Universal Robots URScript: draw_logo.script

def draw_image():
    # Get current TCP pose as starting reference (center of A4 paper)
    pose0 = get_actual_tcp_pose()
    x_c = pose0[0]
    y_c = pose0[1]
    z_c = pose0[2]
    rx  = pose0[3]
    ry  = pose0[4]
    rz  = pose0[5]

    # Movement parameters
    a = 0.3      # acceleration
    v = 0.05     # velocity
    z_lift = 0.01  # lift height between paths

    # A4 paper dimensions: 0.21m x 0.297m
    # SVG dimensions: 268.65231 x 393.11508

    # --- Path segment 1 ---
    # Move to start of segment (pen up)
    movel(p[x_c + -0.029184, y_c + -0.124246, z_c + z_lift, rx, ry, rz], a, v)
    # Lower pen
    movel(p[x_c + -0.029184, y_c + -0.124246, z_c, rx, ry, rz], a, v)

    # Draw path
    movel(p[x_c + -0.029184, y_c + -0.124246, z_c, rx, ry, rz], a, v)
    movel(p[x_c + -0.029184, y_c + -0.124246, z_c, rx, ry, rz], a, v)
    movel(p[x_c + -0.029184, y_c + -0.124246, z_c, rx, ry, rz], a, v)
    movel(p[x_c + -0.029184, y_c + -0.124246, z_c, rx, ry, rz], a, v)
    movel(p[x_c + -0.029184, y_c + -0.124246, z_c, rx, ry, rz], a, v)
    movel(p[x_c + -0.029184, y_c + -0.124246, z_c, rx, ry, rz], a, v)
    movel(p[x_c + -0.029184, y_c + -0.124246, z_c, rx, ry, rz], a, v)
    movel(p[x_c + -0.029184, y_c + -0.124246, z_c, rx, ry, rz], a, v)
    movel(p[x_c + -0.029184, y_c + -0.124246, z_c, rx, ry, rz], a, v)
    movel(p[x_c + -0.029184, y_c + -0.124246, z_c, rx, ry, rz], a, v)
    movel(p[x_c + -0.029182, y_c + -0.124228, z_c, rx, ry, rz], a, v)
    movel(p[x_c + -0.029174, y_c + -0.124205, z_c, rx, ry, rz], a, v)
    movel(p[x_c + -0.029161, y_c + -0.124179, z_c, rx, ry, rz], a, v)
    movel(p[x_c + -0.029143, y_c + -0.124148, z_c, rx, ry, rz], a, v)
    movel(p[x_c + -0.029120, y_c + -0.124114, z_c, rx, ry, rz], a, v)
    movel(p[x_c + -0.029093, y_c + -0.124076, z_c, rx, ry, rz], a, v)
    movel(p[x_c + -0.029062, y_c + -0.124034, z_c, rx, ry, rz], a, v)
    movel(p[x_c + -0.029026, y_c + -0.123989, z_c, rx, ry, rz], a, v)
    movel(p[x_c + -0.028986, y_c + -0.123941, z_c, rx, ry, rz], a, v)
    movel(p[x_c + -0.028943, y_c + -0.123889, z_c, rx, ry, rz], a, v)
    movel(p[x_c + -0.028896, y_c + -0.123835, z_c, rx, ry, rz], a, v)
    movel(p[x_c + -0.028845, y_c + -0.123778, z_c, rx, ry, rz], a, v)
    movel(p[x_c + -0.028791, y_c + -0.123719, z_c, rx, ry, rz], a, v)
    movel(p[x_c + -0.028734, y_c + -0.123657, z_c, rx, ry, rz], a, v)
    movel(p[x_c + -0.028674, y_c + -0.123593, z_c, rx, ry, rz], a, v)
    movel(p[x_c + -0.028610, y_c + -0.123527, z_c, rx, ry, rz], a, v)
    movel(p[x_c + -0.028545, y_c + -0.123459, z_c, rx, ry, rz], a, v)
    movel(p[x_c + -0.028477, y_c + -0.123389, z_c, rx, ry, rz], a, v)
    movel(p[x_c + -0.028406, y_c + -0.123318, z_c, rx, ry, rz], a, v)
    movel(p[x_c + -0.028334, y_c + -0.123245, z_c, rx, ry, rz], a, v)
    movel(p[x_c + -0.028259, y_c + -0.123171, z_c, rx, ry, rz], a, v)
    movel(p[x_c + -0.028183, y_c + -0.123096, z_c, rx, ry, rz], a, v)
    movel(p[x_c + -0.028105, y_c + -0.123021, z_c, rx, ry, rz], a, v)
    movel(p[x_c + -0.028025, y_c + -0.122944, z_c, rx, ry, rz], a, v)
    movel(p[x_c + -0.027945, y_c + -0.122867, z_c, rx, ry, rz], a, v)
    movel(p[x_c + -0.027863, y_c + -0.122789, z_c, rx, ry, rz], a, v)
    movel(p[x_c + -0.027780, y_c + -0.122711, z_c, rx, ry, rz], a, v)
    movel(p[x_c + -0.027697, y_c + -0.122634, z_c, rx, ry, rz], a, v)
    movel(p[x_c + -0.027613, y_c + -0.122556, z_c, rx, ry, rz], a, v)
    movel(p[x_c + -0.027528, y_c + -0.122478, z_c, rx, ry, rz], a, v)
    movel(p[x_c + -0.027444, y_c + -0.122401, z_c, rx, ry, rz], a, v)
    movel(p[x_c + -0.027359, y_c + -0.122324, z_c, rx, ry, rz], a, v)
    movel(p[x_c + -0.027274, y_c + -0.122249, z_c, rx, ry, rz], a, v)
    movel(p[x_c + -0.027190, y_c + -0.122174, z_c, rx, ry, rz], a, v)
    movel(p[x_c + -0.027106, y_c + -0.122100, z_c, rx, ry, rz], a, v)
    movel(p[x_c + -0.027023, y_c + -0.122027, z_c, rx, ry, rz], a, v)
    movel(p[x_c + -0.026940, y_c + -0.121956, z_c, rx, ry, rz], a, v)
    movel(p[x_c + -0.026858, y_c + -0.121886, z_c, rx, ry, rz], a, v)
    movel(p[x_c + -0.026778, y_c + -0.121819, z_c, rx, ry, rz], a, v)
    movel(p[x_c + -0.026699, y_c + -0.121753, z_c, rx, ry, rz], a, v)
    movel(p[x_c + -0.026621, y_c + -0.121689, z_c, rx, ry, rz], a, v)
    movel(p[x_c + -0.026545, y_c + -0.121627, z_c, rx, ry, rz], a, v)
    movel(p[x_c + -0.026471, y_c + -0.121568, z_c, rx, ry, rz], a, v)
    movel(p[x_c + -0.026399, y_c + -0.121511, z_c, rx, ry, rz], a, v)
    movel(p[x_c + -0.026329, y_c + -0.121457, z_c, rx, ry, rz], a, v)
    movel(p[x_c + -0.026261, y_c + -0.121406, z_c, rx, ry, rz], a, v)
    movel(p[x_c + -0.026196, y_c + -0.121357, z_c, rx, ry, rz], a, v)
    movel(p[x_c + -0.026134, y_c + -0.121313, z_c, rx, ry, rz], a, v)
    movel(p[x_c + -0.026074, y_c + -0.121271, z_c, rx, ry, rz], a, v)
    movel(p[x_c + -0.026074, y_c + -0.121271, z_c, rx, ry, rz], a, v)
    movel(p[x_c + -0.025308, y_c + -0.120746, z_c, rx, ry, rz], a, v)
    movel(p[x_c + -0.025308, y_c + -0.120746, z_c, rx, ry, rz], a, v)
    movel(p[x_c + -0.025963, y_c + -0.120548, z_c, rx, ry, rz], a, v)
    movel(p[x_c + -0.025963, y_c + -0.120548, z_c, rx, ry, rz], a, v)
    movel(p[x_c + -0.026039, y_c + -0.120528, z_c, rx, ry, rz], a, v)
    movel(p[x_c + -0.026135, y_c + -0.120508, z_c, rx, ry, rz], a, v)
    movel(p[x_c + -0.026248, y_c + -0.120489, z_c, rx, ry, rz], a, v)
    movel(p[x_c + -0.026379, y_c + -0.120471, z_c, rx, ry, rz], a, v)
    movel(p[x_c + -0.026527, y_c + -0.120453, z_c, rx, ry, rz], a, v)
    movel(p[x_c + -0.026690, y_c + -0.120435, z_c, rx, ry, rz], a, v)
    movel(p[x_c + -0.026869, y_c + -0.120418, z_c, rx, ry, rz], a, v)
    movel(p[x_c + -0.027061, y_c + -0.120402, z_c, rx, ry, rz], a, v)
    movel(p[x_c + -0.027268, y_c + -0.120386, z_c, rx, ry, rz], a, v)
    movel(p[x_c + -0.027487, y_c + -0.120371, z_c, rx, ry, rz], a, v)
    movel(p[x_c + -0.027718, y_c + -0.120357, z_c, rx, ry, rz], a, v)
    movel(p[x_c + -0.027961, y_c + -0.120343, z_c, rx, ry, rz], a, v)
    movel(p[x_c + -0.028214, y_c + -0.120330, z_c, rx, ry, rz], a, v)
    movel(p[x_c + -0.028477, y_c + -0.120317, z_c, rx, ry, rz], a, v)
    movel(p[x_c + -0.028748, y_c + -0.120305, z_c, rx, ry, rz], a, v)
    movel(p[x_c + -0.029028, y_c + -0.120294, z_c, rx, ry, rz], a, v)
    movel(p[x_c + -0.029316, y_c + -0.120283, z_c, rx, ry, rz], a, v)
    movel(p[x_c + -0.029610, y_c + -0.120273, z_c, rx, ry, rz], a, v)
    movel(p[x_c + -0.029910, y_c + -0.120264, z_c, rx, ry, rz], a, v)
    movel(p[x_c + -0.030215, y_c + -0.120255, z_c, rx, ry, rz], a, v)
    movel(p[x_c + -0.030525, y_c + -0.120247, z_c, rx, ry, rz], a, v)
    movel(p[x_c + -0.030838, y_c + -0.120240, z_c, rx, ry, rz], a, v)
    movel(p[x_c + -0.031155, y_c + -0.120234, z_c, rx, ry, rz], a, v)
    movel(p[x_c + -0.031473, y_c + -0.120228, z_c, rx, ry, rz], a, v)
    movel(p[x_c + -0.031793, y_c + -0.120223, z_c, rx, ry, rz], a, v)
    movel(p[x_c + -0.032113, y_c + -0.120219, z_c, rx, ry, rz], a, v)
    movel(p[x_c + -0.032433, y_c + -0.120216, z_c, rx, ry, rz], a, v)
    movel(p[x_c + -0.032752, y_c + -0.120213, z_c, rx, ry, rz], a, v)
    movel(p[x_c + -0.033070, y_c + -0.120212, z_c, rx, ry, rz], a, v)
    movel(p[x_c + -0.033385, y_c + -0.120211, z_c, rx, ry, rz], a, v)
    movel(p[x_c + -0.033697, y_c + -0.120211, z_c, rx, ry, rz], a, v)
    movel(p[x_c + -0.034005, y_c + -0.120211, z_c, rx, ry, rz], a, v)
    movel(p[x_c + -0.034308, y_c + -0.120213, z_c, rx, ry, rz], a, v)
    movel(p[x_c + -0.034605, y_c + -0.120216, z_c, rx, ry, rz], a, v)
    movel(p[x_c + -0.034897, y_c + -0.120219, z_c, rx, ry, rz], a, v)
    movel(p[x_c + -0.035181, y_c + -0.120223, z_c, rx, ry, rz], a, v)
    movel(p[x_c + -0.035458, y_c + -0.120229, z_c, rx, ry, rz], a, v)
    movel(p[x_c + -0.035726, y_c + -0.120235, z_c, rx, ry, rz], a, v)
    movel(p[x_c + -0.035984, y_c + -0.120242, z_c, rx, ry, rz], a, v)
    movel(p[x_c + -0.036233, y_c + -0.120250, z_c, rx, ry, rz], a, v)
    movel(p[x_c + -0.036470, y_c + -0.120259, z_c, rx, ry, rz], a, v)
    movel(p[x_c + -0.036697, y_c + -0.120269, z_c, rx, ry, rz], a, v)
    movel(p[x_c + -0.036910, y_c + -0.120280, z_c, rx, ry, rz], a, v)
    movel(p[x_c + -0.037111, y_c + -0.120291, z_c, rx, ry, rz], a, v)
    movel(p[x_c + -0.037298, y_c + -0.120304, z_c, rx, ry, rz], a, v)
    movel(p[x_c + -0.037470, y_c + -0.120318, z_c, rx, ry, rz], a, v)
    movel(p[x_c + -0.037626, y_c + -0.120333, z_c, rx, ry, rz], a, v)
    movel(p[x_c + -0.037767, y_c + -0.120349, z_c, rx, ry, rz], a, v)
    movel(p[x_c + -0.037890, y_c + -0.120366, z_c, rx, ry, rz], a, v)
    movel(p[x_c + -0.037890, y_c + -0.120366, z_c, rx, ry, rz], a, v)
    movel(p[x_c + -0.038046, y_c + -0.120390, z_c, rx, ry, rz], a, v)
    movel(p[x_c + -0.038202, y_c + -0.120415, z_c, rx, ry, rz], a, v)
    movel(p[x_c + -0.038359, y_c + -0.120441, z_c, rx, ry, rz], a, v)
    movel(p[x_c + -0.038516, y_c + -0.120468, z_c, rx, ry, rz], a, v)
    movel(p[x_c + -0.038673, y_c + -0.120495, z_c, rx, ry, rz], a, v)
    movel(p[x_c + -0.038830, y_c + -0.120523, z_c, rx, ry, rz], a, v)
    movel(p[x_c + -0.038988, y_c + -0.120552, z_c, rx, ry, rz], a, v)
    movel(p[x_c + -0.039146, y_c + -0.120582, z_c, rx, ry, rz], a, v)
    movel(p[x_c + -0.039303, y_c + -0.120612, z_c, rx, ry, rz], a, v)
    movel(p[x_c + -0.039461, y_c + -0.120643, z_c, rx, ry, rz], a, v)
    movel(p[x_c + -0.039618, y_c + -0.120675, z_c, rx, ry, rz], a, v)
    movel(p[x_c + -0.039775, y_c + -0.120707, z_c, rx, ry, rz], a, v)
    movel(p[x_c + -0.039931, y_c + -0.120739, z_c, rx, ry, rz], a, v)
    movel(p[x_c + -0.040086, y_c + -0.120773, z_c, rx, ry, rz], a, v)
    movel(p[x_c + -0.040241, y_c + -0.120807, z_c, rx, ry, rz], a, v)
    movel(p[x_c + -0.040396, y_c + -0.120841, z_c, rx, ry, rz], a, v)
    movel(p[x_c + -0.040549, y_c + -0.120876, z_c, rx, ry, rz], a, v)
    movel(p[x_c + -0.040701, y_c + -0.120911, z_c, rx, ry, rz], a, v)
    movel(p[x_c + -0.040853, y_c + -0.120947, z_c, rx, ry, rz], a, v)
    movel(p[x_c + -0.041003, y_c + -0.120983, z_c, rx, ry, rz], a, v)
    movel(p[x_c + -0.041152, y_c + -0.121019, z_c, rx, ry, rz], a, v)
    movel(p[x_c + -0.041299, y_c + -0.121056, z_c, rx, ry, rz], a, v)
    movel(p[x_c + -0.041445, y_c + -0.121093, z_c, rx, ry, rz], a, v)
    movel(p[x_c + -0.041590, y_c + -0.121131, z_c, rx, ry, rz], a, v)
    movel(p[x_c + -0.041732, y_c + -0.121169, z_c, rx, ry, rz], a, v)
    movel(p[x_c + -0.041874, y_c + -0.121207, z_c, rx, ry, rz], a, v)
    movel(p[x_c + -0.042013, y_c + -0.121245, z_c, rx, ry, rz], a, v)
    movel(p[x_c + -0.042150, y_c + -0.121283, z_c, rx, ry, rz], a, v)
    movel(p[x_c + -0.042285, y_c + -0.121322, z_c, rx, ry, rz], a, v)
    movel(p[x_c + -0.042418, y_c + -0.121360, z_c, rx, ry, rz], a, v)
    movel(p[x_c + -0.042549, y_c + -0.121399, z_c, rx, ry, rz], a, v)
    movel(p[x_c + -0.042678, y_c + -0.121438, z_c, rx, ry, rz], a, v)
    movel(p[x_c + -0.042804, y_c + -0.121477, z_c, rx, ry, rz], a, v)
    movel(p[x_c + -0.042928, y_c + -0.121516, z_c, rx, ry, rz], a, v)
    movel(p[x_c + -0.043049, y_c + -0.121555, z_c, rx, ry, rz], a, v)
    movel(p[x_c + -0.043167, y_c + -0.121594, z_c, rx, ry, rz], a, v)
    movel(p[x_c + -0.043282, y_c + -0.121633, z_c, rx, ry, rz], a, v)
    movel(p[x_c + -0.043395, y_c + -0.121672, z_c, rx, ry, rz], a, v)
    movel(p[x_c + -0.043504, y_c + -0.121711, z_c, rx, ry, rz], a, v)
    movel(p[x_c + -0.043611, y_c + -0.121750, z_c, rx, ry, rz], a, v)
    movel(p[x_c + -0.043714, y_c + -0.121788, z_c, rx, ry, rz], a, v)
    movel(p[x_c + -0.043814, y_c + -0.121827, z_c, rx, ry, rz], a, v)
    movel(p[x_c + -0.043910, y_c + -0.121865, z_c, rx, ry, rz], a, v)
    movel(p[x_c + -0.044003, y_c + -0.121903, z_c, rx, ry, rz], a, v)
    movel(p[x_c + -0.044093, y_c + -0.121940, z_c, rx, ry, rz], a, v)
    movel(p[x_c + -0.044178, y_c + -0.121978, z_c, rx, ry, rz], a, v)
    movel(p[x_c + -0.044260, y_c + -0.122015, z_c, rx, ry, rz], a, v)
    movel(p[x_c + -0.044338, y_c + -0.122052, z_c, rx, ry, rz], a, v)
    movel(p[x_c + -0.044412, y_c + -0.122089, z_c, rx, ry, rz], a, v)
    movel(p[x_c + -0.044412, y_c + -0.122089, z_c, rx, ry, rz], a, v)
    movel(p[x_c + -0.044448, y_c + -0.122106, z_c, rx, ry, rz], a, v)
    movel(p[x_c + -0.044483, y_c + -0.122124, z_c, rx, ry, rz], a, v)
    movel(p[x_c + -0.044518, y_c + -0.122142, z_c, rx, ry, rz], a, v)
    movel(p[x_c + -0.044553, y_c + -0.122159, z_c, rx, ry, rz], a, v)
    movel(p[x_c + -0.044587, y_c + -0.122176, z_c, rx, ry, rz], a, v)
    movel(p[x_c + -0.044622, y_c + -0.122193, z_c, rx, ry, rz], a, v)
    movel(p[x_c + -0.044656, y_c + -0.122210, z_c, rx, ry, rz], a, v)
    movel(p[x_c + -0.044690, y_c + -0.122227, z_c, rx, ry, rz], a, v)
    movel(p[x_c + -0.044723, y_c + -0.122243, z_c, rx, ry, rz], a, v)
    movel(p[x_c + -0.044756, y_c + -0.122259, z_c, rx, ry, rz], a, v)
    movel(p[x_c + -0.044789, y_c + -0.122275, z_c, rx, ry, rz], a, v)
    movel(p[x_c + -0.044822, y_c + -0.122291, z_c, rx, ry, rz], a, v)
    movel(p[x_c + -0.044854, y_c + -0.122307, z_c, rx, ry, rz], a, v)
    movel(p[x_c + -0.044885, y_c + -0.122322, z_c, rx, ry, rz], a, v)
    movel(p[x_c + -0.044917, y_c + -0.122337, z_c, rx, ry, rz], a, v)
    movel(p[x_c + -0.044947, y_c + -0.122351, z_c, rx, ry, rz], a, v)
    movel(p[x_c + -0.044978, y_c + -0.122366, z_c, rx, ry, rz], a, v)
    movel(p[x_c + -0.045007, y_c + -0.122380, z_c, rx, ry, rz], a, v)
    movel(p[x_c + -0.045037, y_c + -0.122394, z_c, rx, ry, rz], a, v)
    movel(p[x_c + -0.045065, y_c + -0.122407, z_c, rx, ry, rz], a, v)
    movel(p[x_c + -0.045094, y_c + -0.122420, z_c, rx, ry, rz], a, v)
    movel(p[x_c + -0.045121, y_c + -0.122433, z_c, rx, ry, rz], a, v)
    movel(p[x_c + -0.045148, y_c + -0.122446, z_c, rx, ry, rz], a, v)
    movel(p[x_c + -0.045175, y_c + -0.122458, z_c, rx, ry, rz], a, v)
    movel(p[x_c + -0.045200, y_c + -0.122470, z_c, rx, ry, rz], a, v)
    movel(p[x_c + -0.045226, y_c + -0.122481, z_c, rx, ry, rz], a, v)
    movel(p[x_c + -0.045250, y_c + -0.122492, z_c, rx, ry, rz], a, v)
    movel(p[x_c + -0.045274, y_c + -0.122503, z_c, rx, ry, rz], a, v)
    movel(p[x_c + -0.045297, y_c + -0.122513, z_c, rx, ry, rz], a, v)
    movel(p[x_c + -0.045319, y_c + -0.122523, z_c, rx, ry, rz], a, v)
    movel(p[x_c + -0.045340, y_c + -0.122532, z_c, rx, ry, rz], a, v)
    movel(p[x_c + -0.045361, y_c + -0.122541, z_c, rx, ry, rz], a, v)
    movel(p[x_c + -0.045381, y_c + -0.122550, z_c, rx, ry, rz], a, v)
    movel(p[x_c + -0.045400, y_c + -0.122558, z_c, rx, ry, rz], a, v)
    movel(p[x_c + -0.045418, y_c + -0.122566, z_c, rx, ry, rz], a, v)
    movel(p[x_c + -0.045436, y_c + -0.122573, z_c, rx, ry, rz], a, v)
    movel(p[x_c + -0.045452, y_c + -0.122580, z_c, rx, ry, rz], a, v)
    movel(p[x_c + -0.045468, y_c + -0.122586, z_c, rx, ry, rz], a, v)
    movel(p[x_c + -0.045482, y_c + -0.122592, z_c, rx, ry, rz], a, v)
    movel(p[x_c + -0.045496, y_c + -0.122597, z_c, rx, ry, rz], a, v)
    movel(p[x_c + -0.045509, y_c + -0.122602, z_c, rx, ry, rz], a, v)
    movel(p[x_c + -0.045520, y_c + -0.122606, z_c, rx, ry, rz], a, v)
    movel(p[x_c + -0.045531, y_c + -0.122610, z_c, rx, ry, rz], a, v)
    movel(p[x_c + -0.045541, y_c + -0.122613, z_c, rx, ry, rz], a, v)
    movel(p[x_c + -0.045549, y_c + -0.122615, z_c, rx, ry, rz], a, v)
    movel(p[x_c + -0.045557, y_c + -0.122617, z_c, rx, ry, rz], a, v)
    movel(p[x_c + -0.045563, y_c + -0.122619, z_c, rx, ry, rz], a, v)
    movel(p[x_c + -0.045569, y_c + -0.122620, z_c, rx, ry, rz], a, v)
    movel(p[x_c + -0.045573, y_c + -0.122620, z_c, rx, ry, rz], a, v)
    movel(p[x_c + -0.045573, y_c + -0.122620, z_c, rx, ry, rz], a, v)
    movel(p[x_c + -0.045587, y_c + -0.122618, z_c, rx, ry, rz], a, v)
    movel(p[x_c + -0.045598, y_c + -0.122613, z_c, rx, ry, rz], a, v)
    movel(p[x_c + -0.045608, y_c + -0.122604, z_c, rx, ry, rz], a, v)
    movel(p[x_c + -0.045615, y_c + -0.122592, z_c, rx, ry, rz], a, v)
    movel(p[x_c + -0.045620, y_c + -0.122576, z_c, rx, ry, rz], a, v)
    movel(p[x_c + -0.045623, y_c + -0.122557, z_c, rx, ry, rz], a, v)
    movel(p[x_c + -0.045623, y_c + -0.122535, z_c, rx, ry, rz], a, v)
    movel(p[x_c + -0.045622, y_c + -0.122509, z_c, rx, ry, rz], a, v)
    movel(p[x_c + -0.045618, y_c + -0.122481, z_c, rx, ry, rz], a, v)
    movel(p[x_c + -0.045613, y_c + -0.122449, z_c, rx, ry, rz], a, v)
    movel(p[x_c + -0.045605, y_c + -0.122414, z_c, rx, ry, rz], a, v)
    movel(p[x_c + -0.045596, y_c + -0.122377, z_c, rx, ry, rz], a, v)
    movel(p[x_c + -0.045584, y_c + -0.122336, z_c, rx, ry, rz], a, v)
    movel(p[x_c + -0.045571, y_c + -0.122293, z_c, rx, ry, rz], a, v)
    movel(p[x_c + -0.045556, y_c + -0.122247, z_c, rx, ry, rz], a, v)
    movel(p[x_c + -0.045539, y_c + -0.122198, z_c, rx, ry, rz], a, v)
    movel(p[x_c + -0.045520, y_c + -0.122147, z_c, rx, ry, rz], a, v)
    movel(p[x_c + -0.045499, y_c + -0.122093, z_c, rx, ry, rz], a, v)
    movel(p[x_c + -0.045476, y_c + -0.122036, z_c, rx, ry, rz], a, v)
    movel(p[x_c + -0.045452, y_c + -0.121977, z_c, rx, ry, rz], a, v)
    movel(p[x_c + -0.045426, y_c + -0.121916, z_c, rx, ry, rz], a, v)
    movel(p[x_c + -0.045398, y_c + -0.121852, z_c, rx, ry, rz], a, v)
    movel(p[x_c + -0.045369, y_c + -0.121786, z_c, rx, ry, rz], a, v)
    movel(p[x_c + -0.045338, y_c + -0.121717, z_c, rx, ry, rz], a, v)
    movel(p[x_c + -0.045305, y_c + -0.121647, z_c, rx, ry, rz], a, v)
    movel(p[x_c + -0.045271, y_c + -0.121574, z_c, rx, ry, rz], a, v)
    movel(p[x_c + -0.045235, y_c + -0.121500, z_c, rx, ry, rz], a, v)
    movel(p[x_c + -0.045198, y_c + -0.121423, z_c, rx, ry, rz], a, v)
    movel(p[x_c + -0.045159, y_c + -0.121345, z_c, rx, ry, rz], a, v)
    movel(p[x_c + -0.045119, y_c + -0.121265, z_c, rx, ry, rz], a, v)
    movel(p[x_c + -0.045077, y_c + -0.121182, z_c, rx, ry, rz], a, v)
    movel(p[x_c + -0.045034, y_c + -0.121099, z_c, rx, ry, rz], a, v)
    movel(p[x_c + -0.044989, y_c + -0.121013, z_c, rx, ry, rz], a, v)
    movel(p[x_c + -0.044943, y_c + -0.120926, z_c, rx, ry, rz], a, v)
    movel(p[x_c + -0.044896, y_c + -0.120837, z_c, rx, ry, rz], a, v)
    movel(p[x_c + -0.044847, y_c + -0.120747, z_c, rx, ry, rz], a, v)
    movel(p[x_c + -0.044798, y_c + -0.120656, z_c, rx, ry, rz], a, v)
    movel(p[x_c + -0.044747, y_c + -0.120563, z_c, rx, ry, rz], a, v)
    movel(p[x_c + -0.044694, y_c + -0.120469, z_c, rx, ry, rz], a, v)
    movel(p[x_c + -0.044641, y_c + -0.120373, z_c, rx, ry, rz], a, v)
    movel(p[x_c + -0.044586, y_c + -0.120276, z_c, rx, ry, rz], a, v)
    movel(p[x_c + -0.044531, y_c + -0.120179, z_c, rx, ry, rz], a, v)
    movel(p[x_c + -0.044474, y_c + -0.120080, z_c, rx, ry, rz], a, v)
    movel(p[x_c + -0.044416, y_c + -0.119980, z_c, rx, ry, rz], a, v)
    movel(p[x_c + -0.044357, y_c + -0.119879, z_c, rx, ry, rz], a, v)
    movel(p[x_c + -0.044297, y_c + -0.119778, z_c, rx, ry, rz], a, v)
    movel(p[x_c + -0.044236, y_c + -0.119675, z_c, rx, ry, rz], a, v)
    movel(p[x_c + -0.044174, y_c + -0.119572, z_c, rx, ry, rz], a, v)
    movel(p[x_c + -0.044111, y_c + -0.119468, z_c, rx, ry, rz], a, v)
    movel(p[x_c + -0.044111, y_c + -0.119468, z_c, rx, ry, rz], a, v)
    movel(p[x_c + -0.044074, y_c + -0.119407, z_c, rx, ry, rz], a, v)
    movel(p[x_c + -0.044038, y_c + -0.119347, z_c, rx, ry, rz], a, v)
    movel(p[x_c + -0.044001, y_c + -0.119286, z_c, rx, ry, rz], a, v)
    movel(p[x_c + -0.043966, y_c + -0.119227, z_c, rx, ry, rz], a, v)
    movel(p[x_c + -0.043930, y_c + -0.119168, z_c, rx, ry, rz], a, v)
    movel(p[x_c + -0.043895, y_c + -0.119109, z_c, rx, ry, rz], a, v)
    movel(p[x_c + -0.043861, y_c + -0.119051, z_c, rx, ry, rz], a, v)
    movel(p[x_c + -0.043827, y_c + -0.118993, z_c, rx, ry, rz], a, v)
    movel(p[x_c + -0.043794, y_c + -0.118936, z_c, rx, ry, rz], a, v)
    movel(p[x_c + -0.043761, y_c + -0.118880, z_c, rx, ry, rz], a, v)
    movel(p[x_c + -0.043729, y_c + -0.118825, z_c, rx, ry, rz], a, v)
    movel(p[x_c + -0.043697, y_c + -0.118770, z_c, rx, ry, rz], a, v)
    movel(p[x_c + -0.043666, y_c + -0.118716, z_c, rx, ry, rz], a, v)
    movel(p[x_c + -0.043635, y_c + -0.118663, z_c, rx, ry, rz], a, v)
    movel(p[x_c + -0.043606, y_c + -0.118610, z_c, rx, ry, rz], a, v)
    movel(p[x_c + -0.043576, y_c + -0.118559, z_c, rx, ry, rz], a, v)
    movel(p[x_c + -0.043548, y_c + -0.118508, z_c, rx, ry, rz], a, v)
    movel(p[x_c + -0.043520, y_c + -0.118459, z_c, rx, ry, rz], a, v)
    movel(p[x_c + -0.043493, y_c + -0.118410, z_c, rx, ry, rz], a, v)
    movel(p[x_c + -0.043466, y_c + -0.118362, z_c, rx, ry, rz], a, v)
    movel(p[x_c + -0.043440, y_c + -0.118316, z_c, rx, ry, rz], a, v)
    movel(p[x_c + -0.043415, y_c + -0.118270, z_c, rx, ry, rz], a, v)
    movel(p[x_c + -0.043391, y_c + -0.118226, z_c, rx, ry, rz], a, v)
    movel(p[x_c + -0.043367, y_c + -0.118182, z_c, rx, ry, rz], a, v)
    movel(p[x_c + -0.043345, y_c + -0.118140, z_c, rx, ry, rz], a, v)
    movel(p[x_c + -0.043323, y_c + -0.118099, z_c, rx, ry, rz], a, v)
    movel(p[x_c + -0.043302, y_c + -0.118060, z_c, rx, ry, rz], a, v)
    movel(p[x_c + -0.043282, y_c + -0.118021, z_c, rx, ry, rz], a, v)
    movel(p[x_c + -0.043263, y_c + -0.117984, z_c, rx, ry, rz], a, v)
    movel(p[x_c + -0.043244, y_c + -0.117948, z_c, rx, ry, rz], a, v)
    movel(p[x_c + -0.043227, y_c + -0.117914, z_c, rx, ry, rz], a, v)
    movel(p[x_c + -0.043210, y_c + -0.117881, z_c, rx, ry, rz], a, v)
    movel(p[x_c + -0.043195, y_c + -0.117849, z_c, rx, ry, rz], a, v)
    movel(p[x_c + -0.043180, y_c + -0.117819, z_c, rx, ry, rz], a, v)
    movel(p[x_c + -0.043166, y_c + -0.117791, z_c, rx, ry, rz], a, v)
    movel(p[x_c + -0.043154, y_c + -0.117764, z_c, rx, ry, rz], a, v)
    movel(p[x_c + -0.043142, y_c + -0.117738, z_c, rx, ry, rz], a, v)
    movel(p[x_c + -0.043132, y_c + -0.117715, z_c, rx, ry, rz], a, v)
    movel(p[x_c + -0.043122, y_c + -0.117692, z_c, rx, ry, rz], a, v)
    movel(p[x_c + -0.043114, y_c + -0.117672, z_c, rx, ry, rz], a, v)
    movel(p[x_c + -0.043107, y_c + -0.117653, z_c, rx, ry, rz], a, v)
    movel(p[x_c + -0.043100, y_c + -0.117636, z_c, rx, ry, rz], a, v)
    movel(p[x_c + -0.043095, y_c + -0.117621, z_c, rx, ry, rz], a, v)
    movel(p[x_c + -0.043091, y_c + -0.117608, z_c, rx, ry, rz], a, v)
    movel(p[x_c + -0.043089, y_c + -0.117596, z_c, rx, ry, rz], a, v)
    movel(p[x_c + -0.043087, y_c + -0.117586, z_c, rx, ry, rz], a, v)
    movel(p[x_c + -0.043087, y_c + -0.117579, z_c, rx, ry, rz], a, v)
    movel(p[x_c + -0.043088, y_c + -0.117573, z_c, rx, ry, rz], a, v)
    movel(p[x_c + -0.043090, y_c + -0.117569, z_c, rx, ry, rz], a, v)
    movel(p[x_c + -0.043090, y_c + -0.117569, z_c, rx, ry, rz], a, v)
    movel(p[x_c + -0.043101, y_c + -0.117562, z_c, rx, ry, rz], a, v)
    movel(p[x_c + -0.043116, y_c + -0.117556, z_c, rx, ry, rz], a, v)
    movel(p[x_c + -0.043136, y_c + -0.117553, z_c, rx, ry, rz], a, v)
    movel(p[x_c + -0.043161, y_c + -0.117551, z_c, rx, ry, rz], a, v)
    movel(p[x_c + -0.043190, y_c + -0.117551, z_c, rx, ry, rz], a, v)
    movel(p[x_c + -0.043223, y_c + -0.117553, z_c, rx, ry, rz], a, v)
    movel(p[x_c + -0.043260, y_c + -0.117557, z_c, rx, ry, rz], a, v)
    movel(p[x_c + -0.043302, y_c + -0.117563, z_c, rx, ry, rz], a, v)
    movel(p[x_c + -0.043347, y_c + -0.117571, z_c, rx, ry, rz], a, v)
    movel(p[x_c + -0.043397, y_c + -0.117580, z_c, rx, ry, rz], a, v)
    movel(p[x_c + -0.043451, y_c + -0.117591, z_c, rx, ry, rz], a, v)
    movel(p[x_c + -0.043508, y_c + -0.117604, z_c, rx, ry, rz], a, v)
    movel(p[x_c + -0.043569, y_c + -0.117618, z_c, rx, ry, rz], a, v)
    movel(p[x_c + -0.043634, y_c + -0.117635, z_c, rx, ry, rz], a, v)
    movel(p[x_c + -0.043702, y_c + -0.117652, z_c, rx, ry, rz], a, v)
    movel(p[x_c + -0.043774, y_c + -0.117672, z_c, rx, ry, rz], a, v)
    movel(p[x_c + -0.043849, y_c + -0.117693, z_c, rx, ry, rz], a, v)
    movel(p[x_c + -0.043928, y_c + -0.117715, z_c, rx, ry, rz], a, v)
    movel(p[x_c + -0.044009, y_c + -0.117739, z_c, rx, ry, rz], a, v)
    movel(p[x_c + -0.044094, y_c + -0.117765, z_c, rx, ry, rz], a, v)
    movel(p[x_c + -0.044182, y_c + -0.117792, z_c, rx, ry, rz], a, v)
    movel(p[x_c + -0.044273, y_c + -0.117820, z_c, rx, ry, rz], a, v)
    movel(p[x_c + -0.044367, y_c + -0.117850, z_c, rx, ry, rz], a, v)
    movel(p[x_c + -0.044464, y_c + -0.117881, z_c, rx, ry, rz], a, v)
    movel(p[x_c + -0.044564, y_c + -0.117913, z_c, rx, ry, rz], a, v)
    movel(p[x_c + -0.044666, y_c + -0.117947, z_c, rx, ry, rz], a, v)
    movel(p[x_c + -0.044770, y_c + -0.117983, z_c, rx, ry, rz], a, v)
    movel(p[x_c + -0.044878, y_c + -0.118019, z_c, rx, ry, rz], a, v)
    movel(p[x_c + -0.044987, y_c + -0.118057, z_c, rx, ry, rz], a, v)
    movel(p[x_c + -0.045099, y_c + -0.118096, z_c, rx, ry, rz], a, v)
    movel(p[x_c + -0.045213, y_c + -0.118136, z_c, rx, ry, rz], a, v)
    movel(p[x_c + -0.045330, y_c + -0.118177, z_c, rx, ry, rz], a, v)
    movel(p[x_c + -0.045448, y_c + -0.118220, z_c, rx, ry, rz], a, v)
    movel(p[x_c + -0.045569, y_c + -0.118263, z_c, rx, ry, rz], a, v)
    movel(p[x_c + -0.045691, y_c + -0.118308, z_c, rx, ry, rz], a, v)
    movel(p[x_c + -0.045816, y_c + -0.118353, z_c, rx, ry, rz], a, v)
    movel(p[x_c + -0.045942, y_c + -0.118400, z_c, rx, ry, rz], a, v)
    movel(p[x_c + -0.046069, y_c + -0.118448, z_c, rx, ry, rz], a, v)
    movel(p[x_c + -0.046199, y_c + -0.118497, z_c, rx, ry, rz], a, v)
    movel(p[x_c + -0.046329, y_c + -0.118546, z_c, rx, ry, rz], a, v)
    movel(p[x_c + -0.046462, y_c + -0.118597, z_c, rx, ry, rz], a, v)
    movel(p[x_c + -0.046595, y_c + -0.118649, z_c, rx, ry, rz], a, v)
    movel(p[x_c + -0.046730, y_c + -0.118701, z_c, rx, ry, rz], a, v)
    movel(p[x_c + -0.046866, y_c + -0.118754, z_c, rx, ry, rz], a, v)
    movel(p[x_c + -0.047003, y_c + -0.118808, z_c, rx, ry, rz], a, v)
    movel(p[x_c + -0.047141, y_c + -0.118863, z_c, rx, ry, rz], a, v)
    movel(p[x_c + -0.047280, y_c + -0.118919, z_c, rx, ry, rz], a, v)
    movel(p[x_c + -0.047420, y_c + -0.118975, z_c, rx, ry, rz], a, v)
    movel(p[x_c + -0.047561, y_c + -0.119032, z_c, rx, ry, rz], a, v)
    movel(p[x_c + -0.047561, y_c + -0.119032, z_c, rx, ry, rz], a, v)
    movel(p[x_c + -0.049754, y_c + -0.119924, z_c, rx, ry, rz], a, v)
    movel(p[x_c + -0.049754, y_c + -0.119924, z_c, rx, ry, rz], a, v)
    movel(p[x_c + -0.049599, y_c + -0.119207, z_c, rx, ry, rz], a, v)
    movel(p[x_c + -0.049599, y_c + -0.119207, z_c, rx, ry, rz], a, v)
    movel(p[x_c + -0.049566, y_c + -0.119070, z_c, rx, ry, rz], a, v)
    movel(p[x_c + -0.049529, y_c + -0.118931, z_c, rx, ry, rz], a, v)
    movel(p[x_c + -0.049485, y_c + -0.118789, z_c, rx, ry, rz], a, v)
    movel(p[x_c + -0.049437, y_c + -0.118645, z_c, rx, ry, rz], a, v)
    movel(p[x_c + -0.049383, y_c + -0.118499, z_c, rx, ry, rz], a, v)
    movel(p[x_c + -0.049324, y_c + -0.118351, z_c, rx, ry, rz], a, v)
    movel(p[x_c + -0.049260, y_c + -0.118202, z_c, rx, ry, rz], a, v)
    movel(p[x_c + -0.049192, y_c + -0.118051, z_c, rx, ry, rz], a, v)
    movel(p[x_c + -0.049118, y_c + -0.117899, z_c, rx, ry, rz], a, v)
    movel(p[x_c + -0.049040, y_c + -0.117746, z_c, rx, ry, rz], a, v)
    movel(p[x_c + -0.048958, y_c + -0.117591, z_c, rx, ry, rz], a, v)
    movel(p[x_c + -0.048871, y_c + -0.117435, z_c, rx, ry, rz], a, v)
    movel(p[x_c + -0.048780, y_c + -0.117279, z_c, rx, ry, rz], a, v)
    movel(p[x_c + -0.048684, y_c + -0.117122, z_c, rx, ry, rz], a, v)
    movel(p[x_c + -0.048585, y_c + -0.116965, z_c, rx, ry, rz], a, v)
    movel(p[x_c + -0.048482, y_c + -0.116807, z_c, rx, ry, rz], a, v)
    movel(p[x_c + -0.048375, y_c + -0.116649, z_c, rx, ry, rz], a, v)
    movel(p[x_c + -0.048264, y_c + -0.116490, z_c, rx, ry, rz], a, v)
    movel(p[x_c + -0.048150, y_c + -0.116332, z_c, rx, ry, rz], a, v)
    movel(p[x_c + -0.048033, y_c + -0.116174, z_c, rx, ry, rz], a, v)
    movel(p[x_c + -0.047912, y_c + -0.116016, z_c, rx, ry, rz], a, v)
    movel(p[x_c + -0.047788, y_c + -0.115859, z_c, rx, ry, rz], a, v)
    movel(p[x_c + -0.047662, y_c + -0.115702, z_c, rx, ry, rz], a, v)
    movel(p[x_c + -0.047532, y_c + -0.115546, z_c, rx, ry, rz], a, v)
    movel(p[x_c + -0.047399, y_c + -0.115391, z_c, rx, ry, rz], a, v)
    movel(p[x_c + -0.047264, y_c + -0.115237, z_c, rx, ry, rz], a, v)
    movel(p[x_c + -0.047126, y_c + -0.115084, z_c, rx, ry, rz], a, v)
    movel(p[x_c + -0.046986, y_c + -0.114933, z_c, rx, ry, rz], a, v)
    movel(p[x_c + -0.046843, y_c + -0.114783, z_c, rx, ry, rz], a, v)
    movel(p[x_c + -0.046699, y_c + -0.114634, z_c, rx, ry, rz], a, v)
    movel(p[x_c + -0.046552, y_c + -0.114487, z_c, rx, ry, rz], a, v)
    movel(p[x_c + -0.046403, y_c + -0.114342, z_c, rx, ry, rz], a, v)
    movel(p[x_c + -0.046252, y_c + -0.114200, z_c, rx, ry, rz], a, v)
    movel(p[x_c + -0.046100, y_c + -0.114059, z_c, rx, ry, rz], a, v)
    movel(p[x_c + -0.045946, y_c + -0.113920, z_c, rx, ry, rz], a, v)
    movel(p[x_c + -0.045791, y_c + -0.113784, z_c, rx, ry, rz], a, v)
    movel(p[x_c + -0.045634, y_c + -0.113651, z_c, rx, ry, rz], a, v)
    movel(p[x_c + -0.045476, y_c + -0.113520, z_c, rx, ry, rz], a, v)
    movel(p[x_c + -0.045317, y_c + -0.113393, z_c, rx, ry, rz], a, v)
    movel(p[x_c + -0.045158, y_c + -0.113268, z_c, rx, ry, rz], a, v)
    movel(p[x_c + -0.044997, y_c + -0.113146, z_c, rx, ry, rz], a, v)
    movel(p[x_c + -0.044835, y_c + -0.113028, z_c, rx, ry, rz], a, v)
    movel(p[x_c + -0.044673, y_c + -0.112913, z_c, rx, ry, rz], a, v)
    movel(p[x_c + -0.044510, y_c + -0.112801, z_c, rx, ry, rz], a, v)
    movel(p[x_c + -0.044347, y_c + -0.112694, z_c, rx, ry, rz], a, v)
    movel(p[x_c + -0.044184, y_c + -0.112590, z_c, rx, ry, rz], a, v)
    movel(p[x_c + -0.044021, y_c + -0.112490, z_c, rx, ry, rz], a, v)
    movel(p[x_c + -0.043857, y_c + -0.112394, z_c, rx, ry, rz], a, v)
    movel(p[x_c + -0.043694, y_c + -0.112303, z_c, rx, ry, rz], a, v)
    movel(p[x_c + -0.043694, y_c + -0.112303, z_c, rx, ry, rz], a, v)
    movel(p[x_c + -0.043598, y_c + -0.112251, z_c, rx, ry, rz], a, v)
    movel(p[x_c + -0.043499, y_c + -0.112199, z_c, rx, ry, rz], a, v)
    movel(p[x_c + -0.043397, y_c + -0.112147, z_c, rx, ry, rz], a, v)
    movel(p[x_c + -0.043293, y_c + -0.112094, z_c, rx, ry, rz], a, v)
    movel(p[x_c + -0.043187, y_c + -0.112042, z_c, rx, ry, rz], a, v)
    movel(p[x_c + -0.043077, y_c + -0.111989, z_c, rx, ry, rz], a, v)
    movel(p[x_c + -0.042966, y_c + -0.111937, z_c, rx, ry, rz], a, v)
    movel(p[x_c + -0.042852, y_c + -0.111884, z_c, rx, ry, rz], a, v)
    movel(p[x_c + -0.042737, y_c + -0.111832, z_c, rx, ry, rz], a, v)
    movel(p[x_c + -0.042619, y_c + -0.111779, z_c, rx, ry, rz], a, v)
    movel(p[x_c + -0.042499, y_c + -0.111727, z_c, rx, ry, rz], a, v)
    movel(p[x_c + -0.042378, y_c + -0.111675, z_c, rx, ry, rz], a, v)
    movel(p[x_c + -0.042255, y_c + -0.111622, z_c, rx, ry, rz], a, v)
    movel(p[x_c + -0.042130, y_c + -0.111571, z_c, rx, ry, rz], a, v)
    movel(p[x_c + -0.042003, y_c + -0.111519, z_c, rx, ry, rz], a, v)
    movel(p[x_c + -0.041876, y_c + -0.111468, z_c, rx, ry, rz], a, v)
    movel(p[x_c + -0.041746, y_c + -0.111417, z_c, rx, ry, rz], a, v)
    movel(p[x_c + -0.041616, y_c + -0.111366, z_c, rx, ry, rz], a, v)
    movel(p[x_c + -0.041484, y_c + -0.111315, z_c, rx, ry, rz], a, v)
    movel(p[x_c + -0.041351, y_c + -0.111266, z_c, rx, ry, rz], a, v)
    movel(p[x_c + -0.041217, y_c + -0.111216, z_c, rx, ry, rz], a, v)
    movel(p[x_c + -0.041083, y_c + -0.111167, z_c, rx, ry, rz], a, v)
    movel(p[x_c + -0.040947, y_c + -0.111118, z_c, rx, ry, rz], a, v)
    movel(p[x_c + -0.040811, y_c + -0.111070, z_c, rx, ry, rz], a, v)
    movel(p[x_c + -0.040674, y_c + -0.111023, z_c, rx, ry, rz], a, v)
    movel(p[x_c + -0.040537, y_c + -0.110976, z_c, rx, ry, rz], a, v)
    movel(p[x_c + -0.040399, y_c + -0.110929, z_c, rx, ry, rz], a, v)
    movel(p[x_c + -0.040261, y_c + -0.110884, z_c, rx, ry, rz], a, v)
    movel(p[x_c + -0.040122, y_c + -0.110839, z_c, rx, ry, rz], a, v)
    movel(p[x_c + -0.039984, y_c + -0.110795, z_c, rx, ry, rz], a, v)
    movel(p[x_c + -0.039845, y_c + -0.110751, z_c, rx, ry, rz], a, v)
    movel(p[x_c + -0.039706, y_c + -0.110708, z_c, rx, ry, rz], a, v)
    movel(p[x_c + -0.039568, y_c + -0.110666, z_c, rx, ry, rz], a, v)
    movel(p[x_c + -0.039430, y_c + -0.110625, z_c, rx, ry, rz], a, v)
    movel(p[x_c + -0.039292, y_c + -0.110585, z_c, rx, ry, rz], a, v)
    movel(p[x_c + -0.039154, y_c + -0.110546, z_c, rx, ry, rz], a, v)
    movel(p[x_c + -0.039017, y_c + -0.110508, z_c, rx, ry, rz], a, v)
    movel(p[x_c + -0.038880, y_c + -0.110470, z_c, rx, ry, rz], a, v)
    movel(p[x_c + -0.038745, y_c + -0.110434, z_c, rx, ry, rz], a, v)
    movel(p[x_c + -0.038609, y_c + -0.110399, z_c, rx, ry, rz], a, v)
    movel(p[x_c + -0.038475, y_c + -0.110364, z_c, rx, ry, rz], a, v)
    movel(p[x_c + -0.038342, y_c + -0.110331, z_c, rx, ry, rz], a, v)
    movel(p[x_c + -0.038210, y_c + -0.110299, z_c, rx, ry, rz], a, v)
    movel(p[x_c + -0.038079, y_c + -0.110269, z_c, rx, ry, rz], a, v)
    movel(p[x_c + -0.037949, y_c + -0.110239, z_c, rx, ry, rz], a, v)
    movel(p[x_c + -0.037821, y_c + -0.110211, z_c, rx, ry, rz], a, v)
    movel(p[x_c + -0.037694, y_c + -0.110184, z_c, rx, ry, rz], a, v)
    movel(p[x_c + -0.037568, y_c + -0.110158, z_c, rx, ry, rz], a, v)
    movel(p[x_c + -0.037444, y_c + -0.110133, z_c, rx, ry, rz], a, v)
    movel(p[x_c + -0.037444, y_c + -0.110133, z_c, rx, ry, rz], a, v)
    movel(p[x_c + -0.037139, y_c + -0.110076, z_c, rx, ry, rz], a, v)
    movel(p[x_c + -0.036822, y_c + -0.110021, z_c, rx, ry, rz], a, v)
    movel(p[x_c + -0.036494, y_c + -0.109967, z_c, rx, ry, rz], a, v)
    movel(p[x_c + -0.036155, y_c + -0.109915, z_c, rx, ry, rz], a, v)
    movel(p[x_c + -0.035807, y_c + -0.109865, z_c, rx, ry, rz], a, v)
    movel(p[x_c + -0.035450, y_c + -0.109817, z_c, rx, ry, rz], a, v)
    movel(p[x_c + -0.035083, y_c + -0.109770, z_c, rx, ry, rz], a, v)
    movel(p[x_c + -0.034708, y_c + -0.109725, z_c, rx, ry, rz], a, v)
    movel(p[x_c + -0.034324, y_c + -0.109682, z_c, rx, ry, rz], a, v)
    movel(p[x_c + -0.033934, y_c + -0.109641, z_c, rx, ry, rz], a, v)
    movel(p[x_c + -0.033536, y_c + -0.109601, z_c, rx, ry, rz], a, v)
    movel(p[x_c + -0.033131, y_c + -0.109563, z_c, rx, ry, rz], a, v)
    movel(p[x_c + -0.032721, y_c + -0.109528, z_c, rx, ry, rz], a, v)
    movel(p[x_c + -0.032305, y_c + -0.109494, z_c, rx, ry, rz], a, v)
    movel(p[x_c + -0.031883, y_c + -0.109462, z_c, rx, ry, rz], a, v)
    movel(p[x_c + -0.031457, y_c + -0.109431, z_c, rx, ry, rz], a, v)
    movel(p[x_c + -0.031027, y_c + -0.109403, z_c, rx, ry, rz], a, v)
    movel(p[x_c + -0.030593, y_c + -0.109377, z_c, rx, ry, rz], a, v)
    movel(p[x_c + -0.030156, y_c + -0.109352, z_c, rx, ry, rz], a, v)
    movel(p[x_c + -0.029716, y_c + -0.109330, z_c, rx, ry, rz], a, v)
    movel(p[x_c + -0.029273, y_c + -0.109309, z_c, rx, ry, rz], a, v)
    movel(p[x_c + -0.028829, y_c + -0.109291, z_c, rx, ry, rz], a, v)
    movel(p[x_c + -0.028384, y_c + -0.109274, z_c, rx, ry, rz], a, v)
    movel(p[x_c + -0.027937, y_c + -0.109259, z_c, rx, ry, rz], a, v)
    movel(p[x_c + -0.027491, y_c + -0.109247, z_c, rx, ry, rz], a, v)
    movel(p[x_c + -0.027044, y_c + -0.109236, z_c, rx, ry, rz], a, v)
    movel(p[x_c + -0.026598, y_c + -0.109228, z_c, rx, ry, rz], a, v)
    movel(p[x_c + -0.026153, y_c + -0.109221, z_c, rx, ry, rz], a, v)
    movel(p[x_c + -0.025710, y_c + -0.109217, z_c, rx, ry, rz], a, v)
    movel(p[x_c + -0.025269, y_c + -0.109214, z_c, rx, ry, rz], a, v)
    movel(p[x_c + -0.024830, y_c + -0.109214, z_c, rx, ry, rz], a, v)
    movel(p[x_c + -0.024394, y_c + -0.109216, z_c, rx, ry, rz], a, v)
    movel(p[x_c + -0.023961, y_c + -0.109220, z_c, rx, ry, rz], a, v)
    movel(p[x_c + -0.023533, y_c + -0.109226, z_c, rx, ry, rz], a, v)
    movel(p[x_c + -0.023109, y_c + -0.109234, z_c, rx, ry, rz], a, v)
    movel(p[x_c + -0.022689, y_c + -0.109244, z_c, rx, ry, rz], a, v)
    movel(p[x_c + -0.022275, y_c + -0.109257, z_c, rx, ry, rz], a, v)
    movel(p[x_c + -0.021867, y_c + -0.109272, z_c, rx, ry, rz], a, v)
    movel(p[x_c + -0.021466, y_c + -0.109289, z_c, rx, ry, rz], a, v)
    movel(p[x_c + -0.021071, y_c + -0.109308, z_c, rx, ry, rz], a, v)
    movel(p[x_c + -0.020683, y_c + -0.109329, z_c, rx, ry, rz], a, v)
    movel(p[x_c + -0.020303, y_c + -0.109353, z_c, rx, ry, rz], a, v)
    movel(p[x_c + -0.019932, y_c + -0.109378, z_c, rx, ry, rz], a, v)
    movel(p[x_c + -0.019569, y_c + -0.109407, z_c, rx, ry, rz], a, v)
    movel(p[x_c + -0.019215, y_c + -0.109437, z_c, rx, ry, rz], a, v)
    movel(p[x_c + -0.018871, y_c + -0.109470, z_c, rx, ry, rz], a, v)
    movel(p[x_c + -0.018537, y_c + -0.109505, z_c, rx, ry, rz], a, v)
    movel(p[x_c + -0.018214, y_c + -0.109542, z_c, rx, ry, rz], a, v)
    movel(p[x_c + -0.017902, y_c + -0.109581, z_c, rx, ry, rz], a, v)
    movel(p[x_c + -0.017902, y_c + -0.109581, z_c, rx, ry, rz], a, v)
    movel(p[x_c + -0.017810, y_c + -0.109594, z_c, rx, ry, rz], a, v)
    movel(p[x_c + -0.017717, y_c + -0.109605, z_c, rx, ry, rz], a, v)
    movel(p[x_c + -0.017625, y_c + -0.109617, z_c, rx, ry, rz], a, v)
    movel(p[x_c + -0.017531, y_c + -0.109628, z_c, rx, ry, rz], a, v)
    movel(p[x_c + -0.017438, y_c + -0.109639, z_c, rx, ry, rz], a, v)
    movel(p[x_c + -0.017344, y_c + -0.109650, z_c, rx, ry, rz], a, v)
    movel(p[x_c + -0.017250, y_c + -0.109661, z_c, rx, ry, rz], a, v)
    movel(p[x_c + -0.017155, y_c + -0.109671, z_c, rx, ry, rz], a, v)
    movel(p[x_c + -0.017061, y_c + -0.109681, z_c, rx, ry, rz], a, v)
    movel(p[x_c + -0.016966, y_c + -0.109690, z_c, rx, ry, rz], a, v)
    movel(p[x_c + -0.016872, y_c + -0.109700, z_c, rx, ry, rz], a, v)
    movel(p[x_c + -0.016777, y_c + -0.109709, z_c, rx, ry, rz], a, v)
    movel(p[x_c + -0.016683, y_c + -0.109718, z_c, rx, ry, rz], a, v)
    movel(p[x_c + -0.016589, y_c + -0.109726, z_c, rx, ry, rz], a, v)
    movel(p[x_c + -0.016495, y_c + -0.109734, z_c, rx, ry, rz], a, v)
    movel(p[x_c + -0.016402, y_c + -0.109742, z_c, rx, ry, rz], a, v)
    movel(p[x_c + -0.016309, y_c + -0.109750, z_c, rx, ry, rz], a, v)
    movel(p[x_c + -0.016217, y_c + -0.109757, z_c, rx, ry, rz], a, v)
    movel(p[x_c + -0.016125, y_c + -0.109764, z_c, rx, ry, rz], a, v)
    movel(p[x_c + -0.016033, y_c + -0.109771, z_c, rx, ry, rz], a, v)
    movel(p[x_c + -0.015943, y_c + -0.109777, z_c, rx, ry, rz], a, v)
    movel(p[x_c + -0.015853, y_c + -0.109783, z_c, rx, ry, rz], a, v)
    movel(p[x_c + -0.015764, y_c + -0.109789, z_c, rx, ry, rz], a, v)
    movel(p[x_c + -0.015675, y_c + -0.109794, z_c, rx, ry, rz], a, v)
    movel(p[x_c + -0.015588, y_c + -0.109799, z_c, rx, ry, rz], a, v)
    movel(p[x_c + -0.015502, y_c + -0.109804, z_c, rx, ry, rz], a, v)
    movel(p[x_c + -0.015416, y_c + -0.109808, z_c, rx, ry, rz], a, v)
    movel(p[x_c + -0.015332, y_c + -0.109812, z_c, rx, ry, rz], a, v)
    movel(p[x_c + -0.015249, y_c + -0.109815, z_c, rx, ry, rz], a, v)
    movel(p[x_c + -0.015168, y_c + -0.109819, z_c, rx, ry, rz], a, v)
    movel(p[x_c + -0.015087, y_c + -0.109821, z_c, rx, ry, rz], a, v)
    movel(p[x_c + -0.015008, y_c + -0.109824, z_c, rx, ry, rz], a, v)
    movel(p[x_c + -0.014931, y_c + -0.109826, z_c, rx, ry, rz], a, v)
    movel(p[x_c + -0.014855, y_c + -0.109828, z_c, rx, ry, rz], a, v)
    movel(p[x_c + -0.014780, y_c + -0.109829, z_c, rx, ry, rz], a, v)
    movel(p[x_c + -0.014707, y_c + -0.109830, z_c, rx, ry, rz], a, v)
    movel(p[x_c + -0.014636, y_c + -0.109831, z_c, rx, ry, rz], a, v)
    movel(p[x_c + -0.014567, y_c + -0.109831, z_c, rx, ry, rz], a, v)
    movel(p[x_c + -0.014499, y_c + -0.109831, z_c, rx, ry, rz], a, v)
    movel(p[x_c + -0.014434, y_c + -0.109831, z_c, rx, ry, rz], a, v)
    movel(p[x_c + -0.014370, y_c + -0.109830, z_c, rx, ry, rz], a, v)
    movel(p[x_c + -0.014309, y_c + -0.109828, z_c, rx, ry, rz], a, v)
    movel(p[x_c + -0.014249, y_c + -0.109827, z_c, rx, ry, rz], a, v)
    movel(p[x_c + -0.014192, y_c + -0.109824, z_c, rx, ry, rz], a, v)
    movel(p[x_c + -0.014137, y_c + -0.109822, z_c, rx, ry, rz], a, v)
    movel(p[x_c + -0.014084, y_c + -0.109819, z_c, rx, ry, rz], a, v)
    movel(p[x_c + -0.014033, y_c + -0.109815, z_c, rx, ry, rz], a, v)
    movel(p[x_c + -0.013985, y_c + -0.109812, z_c, rx, ry, rz], a, v)
    movel(p[x_c + -0.013940, y_c + -0.109807, z_c, rx, ry, rz], a, v)
    movel(p[x_c + -0.013940, y_c + -0.109807, z_c, rx, ry, rz], a, v)
    movel(p[x_c + -0.013862, y_c + -0.109799, z_c, rx, ry, rz], a, v)
    movel(p[x_c + -0.013783, y_c + -0.109789, z_c, rx, ry, rz], a, v)
    movel(p[x_c + -0.013701, y_c + -0.109777, z_c, rx, ry, rz], a, v)
    movel(p[x_c + -0.013617, y_c + -0.109764, z_c, rx, ry, rz], a, v)
    movel(p[x_c + -0.013531, y_c + -0.109749, z_c, rx, ry, rz], a, v)
    movel(p[x_c + -0.013443, y_c + -0.109733, z_c, rx, ry, rz], a, v)
    movel(p[x_c + -0.013354, y_c + -0.109716, z_c, rx, ry, rz], a, v)
    movel(p[x_c + -0.013263, y_c + -0.109698, z_c, rx, ry, rz], a, v)
    movel(p[x_c + -0.013172, y_c + -0.109678, z_c, rx, ry, rz], a, v)
    movel(p[x_c + -0.013079, y_c + -0.109657, z_c, rx, ry, rz], a, v)
    movel(p[x_c + -0.012985, y_c + -0.109635, z_c, rx, ry, rz], a, v)
    movel(p[x_c + -0.012891, y_c + -0.109612, z_c, rx, ry, rz], a, v)
    movel(p[x_c + -0.012796, y_c + -0.109588, z_c, rx, ry, rz], a, v)
    movel(p[x_c + -0.012700, y_c + -0.109563, z_c, rx, ry, rz], a, v)
    movel(p[x_c + -0.012605, y_c + -0.109537, z_c, rx, ry, rz], a, v)
    movel(p[x_c + -0.012509, y_c + -0.109511, z_c, rx, ry, rz], a, v)
    movel(p[x_c + -0.012414, y_c + -0.109483, z_c, rx, ry, rz], a, v)
    movel(p[x_c + -0.012319, y_c + -0.109455, z_c, rx, ry, rz], a, v)
    movel(p[x_c + -0.012224, y_c + -0.109427, z_c, rx, ry, rz], a, v)
    movel(p[x_c + -0.012130, y_c + -0.109397, z_c, rx, ry, rz], a, v)
    movel(p[x_c + -0.012037, y_c + -0.109368, z_c, rx, ry, rz], a, v)
    movel(p[x_c + -0.011945, y_c + -0.109338, z_c, rx, ry, rz], a, v)
    movel(p[x_c + -0.011854, y_c + -0.109307, z_c, rx, ry, rz], a, v)
    movel(p[x_c + -0.011764, y_c + -0.109276, z_c, rx, ry, rz], a, v)
    movel(p[x_c + -0.011676, y_c + -0.109245, z_c, rx, ry, rz], a, v)
    movel(p[x_c + -0.011589, y_c + -0.109214, z_c, rx, ry, rz], a, v)
    movel(p[x_c + -0.011504, y_c + -0.109183, z_c, rx, ry, rz], a, v)
    movel(p[x_c + -0.011421, y_c + -0.109151, z_c, rx, ry, rz], a, v)
    movel(p[x_c + -0.011341, y_c + -0.109119, z_c, rx, ry, rz], a, v)
    movel(p[x_c + -0.011262, y_c + -0.109088, z_c, rx, ry, rz], a, v)
    movel(p[x_c + -0.011186, y_c + -0.109056, z_c, rx, ry, rz], a, v)
    movel(p[x_c + -0.011113, y_c + -0.109025, z_c, rx, ry, rz], a, v)
    movel(p[x_c + -0.011042, y_c + -0.108994, z_c, rx, ry, rz], a, v)
    movel(p[x_c + -0.010975, y_c + -0.108963, z_c, rx, ry, rz], a, v)
    movel(p[x_c + -0.010911, y_c + -0.108933, z_c, rx, ry, rz], a, v)
    movel(p[x_c + -0.010849, y_c + -0.108903, z_c, rx, ry, rz], a, v)
    movel(p[x_c + -0.010792, y_c + -0.108873, z_c, rx, ry, rz], a, v)
    movel(p[x_c + -0.010738, y_c + -0.108844, z_c, rx, ry, rz], a, v)
    movel(p[x_c + -0.010688, y_c + -0.108815, z_c, rx, ry, rz], a, v)
    movel(p[x_c + -0.010642, y_c + -0.108787, z_c, rx, ry, rz], a, v)
    movel(p[x_c + -0.010600, y_c + -0.108760, z_c, rx, ry, rz], a, v)
    movel(p[x_c + -0.010562, y_c + -0.108733, z_c, rx, ry, rz], a, v)
    movel(p[x_c + -0.010529, y_c + -0.108708, z_c, rx, ry, rz], a, v)
    movel(p[x_c + -0.010500, y_c + -0.108683, z_c, rx, ry, rz], a, v)
    movel(p[x_c + -0.010476, y_c + -0.108659, z_c, rx, ry, rz], a, v)
    movel(p[x_c + -0.010458, y_c + -0.108636, z_c, rx, ry, rz], a, v)
    movel(p[x_c + -0.010444, y_c + -0.108614, z_c, rx, ry, rz], a, v)
    movel(p[x_c + -0.010436, y_c + -0.108593, z_c, rx, ry, rz], a, v)
    movel(p[x_c + -0.010433, y_c + -0.108573, z_c, rx, ry, rz], a, v)
    movel(p[x_c + -0.010433, y_c + -0.108573, z_c, rx, ry, rz], a, v)
    movel(p[x_c + -0.010434, y_c + -0.108567, z_c, rx, ry, rz], a, v)
    movel(p[x_c + -0.010436, y_c + -0.108562, z_c, rx, ry, rz], a, v)
    movel(p[x_c + -0.010441, y_c + -0.108555, z_c, rx, ry, rz], a, v)
    movel(p[x_c + -0.010447, y_c + -0.108548, z_c, rx, ry, rz], a, v)
    movel(p[x_c + -0.010455, y_c + -0.108541, z_c, rx, ry, rz], a, v)
    movel(p[x_c + -0.010465, y_c + -0.108533, z_c, rx, ry, rz], a, v)
    movel(p[x_c + -0.010476, y_c + -0.108524, z_c, rx, ry, rz], a, v)
    movel(p[x_c + -0.010489, y_c + -0.108516, z_c, rx, ry, rz], a, v)
    movel(p[x_c + -0.010503, y_c + -0.108506, z_c, rx, ry, rz], a, v)
    movel(p[x_c + -0.010519, y_c + -0.108496, z_c, rx, ry, rz], a, v)
    movel(p[x_c + -0.010537, y_c + -0.108486, z_c, rx, ry, rz], a, v)
    movel(p[x_c + -0.010556, y_c + -0.108476, z_c, rx, ry, rz], a, v)
    movel(p[x_c + -0.010576, y_c + -0.108465, z_c, rx, ry, rz], a, v)
    movel(p[x_c + -0.010598, y_c + -0.108453, z_c, rx, ry, rz], a, v)
    movel(p[x_c + -0.010621, y_c + -0.108442, z_c, rx, ry, rz], a, v)
    movel(p[x_c + -0.010646, y_c + -0.108430, z_c, rx, ry, rz], a, v)
    movel(p[x_c + -0.010672, y_c + -0.108417, z_c, rx, ry, rz], a, v)
    movel(p[x_c + -0.010700, y_c + -0.108404, z_c, rx, ry, rz], a, v)
    movel(p[x_c + -0.010728, y_c + -0.108391, z_c, rx, ry, rz], a, v)
    movel(p[x_c + -0.010758, y_c + -0.108378, z_c, rx, ry, rz], a, v)
    movel(p[x_c + -0.010790, y_c + -0.108364, z_c, rx, ry, rz], a, v)
    movel(p[x_c + -0.010822, y_c + -0.108350, z_c, rx, ry, rz], a, v)
    movel(p[x_c + -0.010856, y_c + -0.108336, z_c, rx, ry, rz], a, v)
    movel(p[x_c + -0.010890, y_c + -0.108321, z_c, rx, ry, rz], a, v)
    movel(p[x_c + -0.010926, y_c + -0.108306, z_c, rx, ry, rz], a, v)
    movel(p[x_c + -0.010963, y_c + -0.108291, z_c, rx, ry, rz], a, v)
    movel(p[x_c + -0.011001, y_c + -0.108276, z_c, rx, ry, rz], a, v)
    movel(p[x_c + -0.011041, y_c + -0.108260, z_c, rx, ry, rz], a, v)
    movel(p[x_c + -0.011081, y_c + -0.108244, z_c, rx, ry, rz], a, v)
    movel(p[x_c + -0.011122, y_c + -0.108228, z_c, rx, ry, rz], a, v)
    movel(p[x_c + -0.011164, y_c + -0.108212, z_c, rx, ry, rz], a, v)
    movel(p[x_c + -0.011207, y_c + -0.108196, z_c, rx, ry, rz], a, v)
    movel(p[x_c + -0.011251, y_c + -0.108179, z_c, rx, ry, rz], a, v)
    movel(p[x_c + -0.011295, y_c + -0.108163, z_c, rx, ry, rz], a, v)
    movel(p[x_c + -0.011341, y_c + -0.108146, z_c, rx, ry, rz], a, v)
    movel(p[x_c + -0.011387, y_c + -0.108129, z_c, rx, ry, rz], a, v)
    movel(p[x_c + -0.011435, y_c + -0.108112, z_c, rx, ry, rz], a, v)
    movel(p[x_c + -0.011483, y_c + -0.108095, z_c, rx, ry, rz], a, v)
    movel(p[x_c + -0.011531, y_c + -0.108078, z_c, rx, ry, rz], a, v)
    movel(p[x_c + -0.011581, y_c + -0.108060, z_c, rx, ry, rz], a, v)
    movel(p[x_c + -0.011631, y_c + -0.108043, z_c, rx, ry, rz], a, v)
    movel(p[x_c + -0.011681, y_c + -0.108026, z_c, rx, ry, rz], a, v)
    movel(p[x_c + -0.011732, y_c + -0.108008, z_c, rx, ry, rz], a, v)
    movel(p[x_c + -0.011784, y_c + -0.107991, z_c, rx, ry, rz], a, v)
    movel(p[x_c + -0.011837, y_c + -0.107973, z_c, rx, ry, rz], a, v)
    movel(p[x_c + -0.011889, y_c + -0.107956, z_c, rx, ry, rz], a, v)
    movel(p[x_c + -0.011943, y_c + -0.107938, z_c, rx, ry, rz], a, v)
    movel(p[x_c + -0.011997, y_c + -0.107921, z_c, rx, ry, rz], a, v)
    movel(p[x_c + -0.012051, y_c + -0.107903, z_c, rx, ry, rz], a, v)
    movel(p[x_c + -0.012051, y_c + -0.107903, z_c, rx, ry, rz], a, v)
    movel(p[x_c + -0.012260, y_c + -0.107835, z_c, rx, ry, rz], a, v)
    movel(p[x_c + -0.012469, y_c + -0.107765, z_c, rx, ry, rz], a, v)
    movel(p[x_c + -0.012678, y_c + -0.107693, z_c, rx, ry, rz], a, v)
    movel(p[x_c + -0.012888, y_c + -0.107619, z_c, rx, ry, rz], a, v)
    movel(p[x_c + -0.013097, y_c + -0.107542, z_c, rx, ry, rz], a, v)
    movel(p[x_c + -0.013307, y_c + -0.107463, z_c, rx, ry, rz], a, v)
    movel(p[x_c + -0.013516, y_c + -0.107382, z_c, rx, ry, rz], a, v)
    movel(p[x_c + -0.013725, y_c + -0.107299, z_c, rx, ry, rz], a, v)
    movel(p[x_c + -0.013935, y_c + -0.107214, z_c, rx, ry, rz], a, v)
    movel(p[x_c + -0.014144, y_c + -0.107127, z_c, rx, ry, rz], a, v)
    movel(p[x_c + -0.014353, y_c + -0.107038, z_c, rx, ry, rz], a, v)
    movel(p[x_c + -0.014561, y_c + -0.106946, z_c, rx, ry, rz], a, v)
    movel(p[x_c + -0.014770, y_c + -0.106853, z_c, rx, ry, rz], a, v)
    movel(p[x_c + -0.014978, y_c + -0.106758, z_c, rx, ry, rz], a, v)
    movel(p[x_c + -0.015186, y_c + -0.106661, z_c, rx, ry, rz], a, v)
    movel(p[x_c + -0.015393, y_c + -0.106562, z_c, rx, ry, rz], a, v)
    movel(p[x_c + -0.015600, y_c + -0.106461, z_c, rx, ry, rz], a, v)
    movel(p[x_c + -0.015807, y_c + -0.106359, z_c, rx, ry, rz], a, v)
    movel(p[x_c + -0.016013, y_c + -0.106254, z_c, rx, ry, rz], a, v)
    movel(p[x_c + -0.016218, y_c + -0.106148, z_c, rx, ry, rz], a, v)
    movel(p[x_c + -0.016423, y_c + -0.106039, z_c, rx, ry, rz], a, v)
    movel(p[x_c + -0.016627, y_c + -0.105929, z_c, rx, ry, rz], a, v)
    movel(p[x_c + -0.016831, y_c + -0.105818, z_c, rx, ry, rz], a, v)
    movel(p[x_c + -0.017034, y_c + -0.105704, z_c, rx, ry, rz], a, v)
    movel(p[x_c + -0.017236, y_c + -0.105589, z_c, rx, ry, rz], a, v)
    movel(p[x_c + -0.017437, y_c + -0.105472, z_c, rx, ry, rz], a, v)
    movel(p[x_c + -0.017638, y_c + -0.105354, z_c, rx, ry, rz], a, v)
    movel(p[x_c + -0.017838, y_c + -0.105234, z_c, rx, ry, rz], a, v)
    movel(p[x_c + -0.018036, y_c + -0.105112, z_c, rx, ry, rz], a, v)
    movel(p[x_c + -0.018234, y_c + -0.104989, z_c, rx, ry, rz], a, v)
    movel(p[x_c + -0.018431, y_c + -0.104864, z_c, rx, ry, rz], a, v)
    movel(p[x_c + -0.018627, y_c + -0.104737, z_c, rx, ry, rz], a, v)
    movel(p[x_c + -0.018822, y_c + -0.104609, z_c, rx, ry, rz], a, v)
    movel(p[x_c + -0.019015, y_c + -0.104480, z_c, rx, ry, rz], a, v)
    movel(p[x_c + -0.019208, y_c + -0.104349, z_c, rx, ry, rz], a, v)
    movel(p[x_c + -0.019399, y_c + -0.104216, z_c, rx, ry, rz], a, v)
    movel(p[x_c + -0.019589, y_c + -0.104083, z_c, rx, ry, rz], a, v)
    movel(p[x_c + -0.019778, y_c + -0.103947, z_c, rx, ry, rz], a, v)
    movel(p[x_c + -0.019965, y_c + -0.103811, z_c, rx, ry, rz], a, v)
    movel(p[x_c + -0.020152, y_c + -0.103673, z_c, rx, ry, rz], a, v)
    movel(p[x_c + -0.020336, y_c + -0.103533, z_c, rx, ry, rz], a, v)
    movel(p[x_c + -0.020520, y_c + -0.103393, z_c, rx, ry, rz], a, v)
    movel(p[x_c + -0.020702, y_c + -0.103251, z_c, rx, ry, rz], a, v)
    movel(p[x_c + -0.020882, y_c + -0.103108, z_c, rx, ry, rz], a, v)
    movel(p[x_c + -0.021061, y_c + -0.102963, z_c, rx, ry, rz], a, v)
    movel(p[x_c + -0.021238, y_c + -0.102818, z_c, rx, ry, rz], a, v)
    movel(p[x_c + -0.021414, y_c + -0.102671, z_c, rx, ry, rz], a, v)
    movel(p[x_c + -0.021588, y_c + -0.102523, z_c, rx, ry, rz], a, v)
    movel(p[x_c + -0.021760, y_c + -0.102373, z_c, rx, ry, rz], a, v)
    movel(p[x_c + -0.021760, y_c + -0.102373, z_c, rx, ry, rz], a, v)
    movel(p[x_c + -0.021949, y_c + -0.102205, z_c, rx, ry, rz], a, v)
    movel(p[x_c + -0.022137, y_c + -0.102033, z_c, rx, ry, rz], a, v)
    movel(p[x_c + -0.022324, y_c + -0.101856, z_c, rx, ry, rz], a, v)
    movel(p[x_c + -0.022510, y_c + -0.101675, z_c, rx, ry, rz], a, v)
    movel(p[x_c + -0.022695, y_c + -0.101490, z_c, rx, ry, rz], a, v)
    movel(p[x_c + -0.022878, y_c + -0.101300, z_c, rx, ry, rz], a, v)
    movel(p[x_c + -0.023061, y_c + -0.101107, z_c, rx, ry, rz], a, v)
    movel(p[x_c + -0.023242, y_c + -0.100909, z_c, rx, ry, rz], a, v)
    movel(p[x_c + -0.023422, y_c + -0.100706, z_c, rx, ry, rz], a, v)
    movel(p[x_c + -0.023601, y_c + -0.100500, z_c, rx, ry, rz], a, v)
    movel(p[x_c + -0.023778, y_c + -0.100290, z_c, rx, ry, rz], a, v)
    movel(p[x_c + -0.023954, y_c + -0.100075, z_c, rx, ry, rz], a, v)
    movel(p[x_c + -0.024129, y_c + -0.099856, z_c, rx, ry, rz], a, v)
    movel(p[x_c + -0.024303, y_c + -0.099633, z_c, rx, ry, rz], a, v)
    movel(p[x_c + -0.024476, y_c + -0.099406, z_c, rx, ry, rz], a, v)
    movel(p[x_c + -0.024647, y_c + -0.099175, z_c, rx, ry, rz], a, v)
    movel(p[x_c + -0.024817, y_c + -0.098940, z_c, rx, ry, rz], a, v)
    movel(p[x_c + -0.024985, y_c + -0.098701, z_c, rx, ry, rz], a, v)
    movel(p[x_c + -0.025153, y_c + -0.098457, z_c, rx, ry, rz], a, v)
    movel(p[x_c + -0.025319, y_c + -0.098210, z_c, rx, ry, rz], a, v)
    movel(p[x_c + -0.025484, y_c + -0.097959, z_c, rx, ry, rz], a, v)
    movel(p[x_c + -0.025647, y_c + -0.097703, z_c, rx, ry, rz], a, v)
    movel(p[x_c + -0.025809, y_c + -0.097444, z_c, rx, ry, rz], a, v)
    movel(p[x_c + -0.025970, y_c + -0.097181, z_c, rx, ry, rz], a, v)
    movel(p[x_c + -0.026129, y_c + -0.096914, z_c, rx, ry, rz], a, v)
    movel(p[x_c + -0.026287, y_c + -0.096643, z_c, rx, ry, rz], a, v)
    movel(p[x_c + -0.026444, y_c + -0.096368, z_c, rx, ry, rz], a, v)
    movel(p[x_c + -0.026599, y_c + -0.096089, z_c, rx, ry, rz], a, v)
    movel(p[x_c + -0.026753, y_c + -0.095806, z_c, rx, ry, rz], a, v)
    movel(p[x_c + -0.026905, y_c + -0.095519, z_c, rx, ry, rz], a, v)
    movel(p[x_c + -0.027056, y_c + -0.095229, z_c, rx, ry, rz], a, v)
    movel(p[x_c + -0.027206, y_c + -0.094934, z_c, rx, ry, rz], a, v)
    movel(p[x_c + -0.027354, y_c + -0.094636, z_c, rx, ry, rz], a, v)
    movel(p[x_c + -0.027501, y_c + -0.094334, z_c, rx, ry, rz], a, v)
    movel(p[x_c + -0.027646, y_c + -0.094028, z_c, rx, ry, rz], a, v)
    movel(p[x_c + -0.027790, y_c + -0.093719, z_c, rx, ry, rz], a, v)
    movel(p[x_c + -0.027933, y_c + -0.093405, z_c, rx, ry, rz], a, v)
    movel(p[x_c + -0.028073, y_c + -0.093088, z_c, rx, ry, rz], a, v)
    movel(p[x_c + -0.028213, y_c + -0.092767, z_c, rx, ry, rz], a, v)
    movel(p[x_c + -0.028351, y_c + -0.092443, z_c, rx, ry, rz], a, v)
    movel(p[x_c + -0.028487, y_c + -0.092115, z_c, rx, ry, rz], a, v)
    movel(p[x_c + -0.028622, y_c + -0.091783, z_c, rx, ry, rz], a, v)
    movel(p[x_c + -0.028755, y_c + -0.091447, z_c, rx, ry, rz], a, v)
    movel(p[x_c + -0.028887, y_c + -0.091108, z_c, rx, ry, rz], a, v)
    movel(p[x_c + -0.029017, y_c + -0.090765, z_c, rx, ry, rz], a, v)
    movel(p[x_c + -0.029146, y_c + -0.090419, z_c, rx, ry, rz], a, v)
    movel(p[x_c + -0.029273, y_c + -0.090069, z_c, rx, ry, rz], a, v)
    movel(p[x_c + -0.029399, y_c + -0.089715, z_c, rx, ry, rz], a, v)
    movel(p[x_c + -0.029523, y_c + -0.089358, z_c, rx, ry, rz], a, v)
    movel(p[x_c + -0.029523, y_c + -0.089358, z_c, rx, ry, rz], a, v)
    movel(p[x_c + -0.029613, y_c + -0.089097, z_c, rx, ry, rz], a, v)
    movel(p[x_c + -0.029701, y_c + -0.088842, z_c, rx, ry, rz], a, v)
    movel(p[x_c + -0.029789, y_c + -0.088593, z_c, rx, ry, rz], a, v)
    movel(p[x_c + -0.029875, y_c + -0.088350, z_c, rx, ry, rz], a, v)
    movel(p[x_c + -0.029961, y_c + -0.088112, z_c, rx, ry, rz], a, v)
    movel(p[x_c + -0.030046, y_c + -0.087879, z_c, rx, ry, rz], a, v)
    movel(p[x_c + -0.030130, y_c + -0.087651, z_c, rx, ry, rz], a, v)
    movel(p[x_c + -0.030214, y_c + -0.087427, z_c, rx, ry, rz], a, v)
    movel(p[x_c + -0.030298, y_c + -0.087207, z_c, rx, ry, rz], a, v)
    movel(p[x_c + -0.030382, y_c + -0.086991, z_c, rx, ry, rz], a, v)
    movel(p[x_c + -0.030466, y_c + -0.086778, z_c, rx, ry, rz], a, v)
    movel(p[x_c + -0.030550, y_c + -0.086569, z_c, rx, ry, rz], a, v)
    movel(p[x_c + -0.030634, y_c + -0.086362, z_c, rx, ry, rz], a, v)
    movel(p[x_c + -0.030719, y_c + -0.086158, z_c, rx, ry, rz], a, v)
    movel(p[x_c + -0.030805, y_c + -0.085956, z_c, rx, ry, rz], a, v)
    movel(p[x_c + -0.030892, y_c + -0.085756, z_c, rx, ry, rz], a, v)
    movel(p[x_c + -0.030980, y_c + -0.085558, z_c, rx, ry, rz], a, v)
    movel(p[x_c + -0.031069, y_c + -0.085361, z_c, rx, ry, rz], a, v)
    movel(p[x_c + -0.031160, y_c + -0.085165, z_c, rx, ry, rz], a, v)
    movel(p[x_c + -0.031252, y_c + -0.084969, z_c, rx, ry, rz], a, v)
    movel(p[x_c + -0.031346, y_c + -0.084774, z_c, rx, ry, rz], a, v)
    movel(p[x_c + -0.031441, y_c + -0.084579, z_c, rx, ry, rz], a, v)
    movel(p[x_c + -0.031539, y_c + -0.084384, z_c, rx, ry, rz], a, v)
    movel(p[x_c + -0.031639, y_c + -0.084188, z_c, rx, ry, rz], a, v)
    movel(p[x_c + -0.031741, y_c + -0.083991, z_c, rx, ry, rz], a, v)
    movel(p[x_c + -0.031846, y_c + -0.083793, z_c, rx, ry, rz], a, v)
    movel(p[x_c + -0.031954, y_c + -0.083593, z_c, rx, ry, rz], a, v)
    movel(p[x_c + -0.032064, y_c + -0.083392, z_c, rx, ry, rz], a, v)
    movel(p[x_c + -0.032178, y_c + -0.083189, z_c, rx, ry, rz], a, v)
    movel(p[x_c + -0.032294, y_c + -0.082983, z_c, rx, ry, rz], a, v)
    movel(p[x_c + -0.032414, y_c + -0.082774, z_c, rx, ry, rz], a, v)
    movel(p[x_c + -0.032537, y_c + -0.082562, z_c, rx, ry, rz], a, v)
    movel(p[x_c + -0.032665, y_c + -0.082347, z_c, rx, ry, rz], a, v)
    movel(p[x_c + -0.032795, y_c + -0.082129, z_c, rx, ry, rz], a, v)
    movel(p[x_c + -0.032930, y_c + -0.081906, z_c, rx, ry, rz], a, v)
    movel(p[x_c + -0.033069, y_c + -0.081679, z_c, rx, ry, rz], a, v)
    movel(p[x_c + -0.033212, y_c + -0.081447, z_c, rx, ry, rz], a, v)
    movel(p[x_c + -0.033360, y_c + -0.081211, z_c, rx, ry, rz], a, v)
    movel(p[x_c + -0.033513, y_c + -0.080969, z_c, rx, ry, rz], a, v)
    movel(p[x_c + -0.033670, y_c + -0.080722, z_c, rx, ry, rz], a, v)
    movel(p[x_c + -0.033832, y_c + -0.080469, z_c, rx, ry, rz], a, v)
    movel(p[x_c + -0.033999, y_c + -0.080209, z_c, rx, ry, rz], a, v)
    movel(p[x_c + -0.034171, y_c + -0.079944, z_c, rx, ry, rz], a, v)
    movel(p[x_c + -0.034349, y_c + -0.079671, z_c, rx, ry, rz], a, v)
    movel(p[x_c + -0.034533, y_c + -0.079392, z_c, rx, ry, rz], a, v)
    movel(p[x_c + -0.034722, y_c + -0.079105, z_c, rx, ry, rz], a, v)
    movel(p[x_c + -0.034917, y_c + -0.078810, z_c, rx, ry, rz], a, v)
    movel(p[x_c + -0.035118, y_c + -0.078507, z_c, rx, ry, rz], a, v)
    movel(p[x_c + -0.035325, y_c + -0.078196, z_c, rx, ry, rz], a, v)
    movel(p[x_c + -0.035325, y_c + -0.078196, z_c, rx, ry, rz], a, v)
    movel(p[x_c + -0.035567, y_c + -0.077835, z_c, rx, ry, rz], a, v)
    movel(p[x_c + -0.035802, y_c + -0.077481, z_c, rx, ry, rz], a, v)
    movel(p[x_c + -0.036032, y_c + -0.077135, z_c, rx, ry, rz], a, v)
    movel(p[x_c + -0.036256, y_c + -0.076797, z_c, rx, ry, rz], a, v)
    movel(p[x_c + -0.036475, y_c + -0.076465, z_c, rx, ry, rz], a, v)
    movel(p[x_c + -0.036689, y_c + -0.076141, z_c, rx, ry, rz], a, v)
    movel(p[x_c + -0.036897, y_c + -0.075823, z_c, rx, ry, rz], a, v)
    movel(p[x_c + -0.037101, y_c + -0.075511, z_c, rx, ry, rz], a, v)
    movel(p[x_c + -0.037300, y_c + -0.075205, z_c, rx, ry, rz], a, v)
    movel(p[x_c + -0.037494, y_c + -0.074905, z_c, rx, ry, rz], a, v)
    movel(p[x_c + -0.037684, y_c + -0.074611, z_c, rx, ry, rz], a, v)
    movel(p[x_c + -0.037870, y_c + -0.074322, z_c, rx, ry, rz], a, v)
    movel(p[x_c + -0.038051, y_c + -0.074038, z_c, rx, ry, rz], a, v)
    movel(p[x_c + -0.038229, y_c + -0.073758, z_c, rx, ry, rz], a, v)
    movel(p[x_c + -0.038403, y_c + -0.073483, z_c, rx, ry, rz], a, v)
    movel(p[x_c + -0.038573, y_c + -0.073213, z_c, rx, ry, rz], a, v)
    movel(p[x_c + -0.038740, y_c + -0.072945, z_c, rx, ry, rz], a, v)
    movel(p[x_c + -0.038904, y_c + -0.072682, z_c, rx, ry, rz], a, v)
    movel(p[x_c + -0.039064, y_c + -0.072422, z_c, rx, ry, rz], a, v)
    movel(p[x_c + -0.039222, y_c + -0.072165, z_c, rx, ry, rz], a, v)
    movel(p[x_c + -0.039376, y_c + -0.071910, z_c, rx, ry, rz], a, v)
    movel(p[x_c + -0.039528, y_c + -0.071659, z_c, rx, ry, rz], a, v)
    movel(p[x_c + -0.039678, y_c + -0.071409, z_c, rx, ry, rz], a, v)
    movel(p[x_c + -0.039825, y_c + -0.071161, z_c, rx, ry, rz], a, v)
    movel(p[x_c + -0.039971, y_c + -0.070915, z_c, rx, ry, rz], a, v)
    movel(p[x_c + -0.040114, y_c + -0.070671, z_c, rx, ry, rz], a, v)
    movel(p[x_c + -0.040255, y_c + -0.070427, z_c, rx, ry, rz], a, v)
    movel(p[x_c + -0.040395, y_c + -0.070185, z_c, rx, ry, rz], a, v)
    movel(p[x_c + -0.040533, y_c + -0.069943, z_c, rx, ry, rz], a, v)
    movel(p[x_c + -0.040670, y_c + -0.069701, z_c, rx, ry, rz], a, v)
    movel(p[x_c + -0.040805, y_c + -0.069459, z_c, rx, ry, rz], a, v)
    movel(p[x_c + -0.040940, y_c + -0.069217, z_c, rx, ry, rz], a, v)
    movel(p[x_c + -0.041074, y_c + -0.068975, z_c, rx, ry, rz], a, v)
    movel(p[x_c + -0.041207, y_c + -0.068732, z_c, rx, ry, rz], a, v)
    movel(p[x_c + -0.041339, y_c + -0.068487, z_c, rx, ry, rz], a, v)
    movel(p[x_c + -0.041471, y_c + -0.068242, z_c, rx, ry, rz], a, v)
    movel(p[x_c + -0.041603, y_c + -0.067994, z_c, rx, ry, rz], a, v)
    movel(p[x_c + -0.041735, y_c + -0.067745, z_c, rx, ry, rz], a, v)
    movel(p[x_c + -0.041867, y_c + -0.067494, z_c, rx, ry, rz], a, v)
    movel(p[x_c + -0.041999, y_c + -0.067240, z_c, rx, ry, rz], a, v)
    movel(p[x_c + -0.042132, y_c + -0.066984, z_c, rx, ry, rz], a, v)
    movel(p[x_c + -0.042265, y_c + -0.066725, z_c, rx, ry, rz], a, v)
    movel(p[x_c + -0.042399, y_c + -0.066462, z_c, rx, ry, rz], a, v)
    movel(p[x_c + -0.042534, y_c + -0.066196, z_c, rx, ry, rz], a, v)
    movel(p[x_c + -0.042670, y_c + -0.065926, z_c, rx, ry, rz], a, v)
    movel(p[x_c + -0.042808, y_c + -0.065652, z_c, rx, ry, rz], a, v)
    movel(p[x_c + -0.042946, y_c + -0.065374, z_c, rx, ry, rz], a, v)
    movel(p[x_c + -0.043086, y_c + -0.065091, z_c, rx, ry, rz], a, v)
    movel(p[x_c + -0.043228, y_c + -0.064803, z_c, rx, ry, rz], a, v)
    movel(p[x_c + -0.043228, y_c + -0.064803, z_c, rx, ry, rz], a, v)
    movel(p[x_c + -0.043407, y_c + -0.064438, z_c, rx, ry, rz], a, v)
    movel(p[x_c + -0.043583, y_c + -0.064075, z_c, rx, ry, rz], a, v)
    movel(p[x_c + -0.043757, y_c + -0.063713, z_c, rx, ry, rz], a, v)
    movel(p[x_c + -0.043929, y_c + -0.063351, z_c, rx, ry, rz], a, v)
    movel(p[x_c + -0.044099, y_c + -0.062990, z_c, rx, ry, rz], a, v)
    movel(p[x_c + -0.044267, y_c + -0.062630, z_c, rx, ry, rz], a, v)
    movel(p[x_c + -0.044433, y_c + -0.062271, z_c, rx, ry, rz], a, v)
    movel(p[x_c + -0.044597, y_c + -0.061913, z_c, rx, ry, rz], a, v)
    movel(p[x_c + -0.044759, y_c + -0.061555, z_c, rx, ry, rz], a, v)
    movel(p[x_c + -0.044918, y_c + -0.061198, z_c, rx, ry, rz], a, v)
    movel(p[x_c + -0.045076, y_c + -0.060841, z_c, rx, ry, rz], a, v)
    movel(p[x_c + -0.045232, y_c + -0.060485, z_c, rx, ry, rz], a, v)
    movel(p[x_c + -0.045386, y_c + -0.060130, z_c, rx, ry, rz], a, v)
    movel(p[x_c + -0.045537, y_c + -0.059775, z_c, rx, ry, rz], a, v)
    movel(p[x_c + -0.045687, y_c + -0.059420, z_c, rx, ry, rz], a, v)
    movel(p[x_c + -0.045835, y_c + -0.059066, z_c, rx, ry, rz], a, v)
    movel(p[x_c + -0.045981, y_c + -0.058712, z_c, rx, ry, rz], a, v)
    movel(p[x_c + -0.046126, y_c + -0.058358, z_c, rx, ry, rz], a, v)
    movel(p[x_c + -0.046268, y_c + -0.058005, z_c, rx, ry, rz], a, v)
    movel(p[x_c + -0.046408, y_c + -0.057652, z_c, rx, ry, rz], a, v)
    movel(p[x_c + -0.046547, y_c + -0.057299, z_c, rx, ry, rz], a, v)
    movel(p[x_c + -0.046684, y_c + -0.056946, z_c, rx, ry, rz], a, v)
    movel(p[x_c + -0.046819, y_c + -0.056593, z_c, rx, ry, rz], a, v)
    movel(p[x_c + -0.046952, y_c + -0.056240, z_c, rx, ry, rz], a, v)
    movel(p[x_c + -0.047084, y_c + -0.055887, z_c, rx, ry, rz], a, v)
    movel(p[x_c + -0.047213, y_c + -0.055534, z_c, rx, ry, rz], a, v)
    movel(p[x_c + -0.047341, y_c + -0.055180, z_c, rx, ry, rz], a, v)
    movel(p[x_c + -0.047468, y_c + -0.054827, z_c, rx, ry, rz], a, v)
    movel(p[x_c + -0.047592, y_c + -0.054473, z_c, rx, ry, rz], a, v)
    movel(p[x_c + -0.047715, y_c + -0.054120, z_c, rx, ry, rz], a, v)
    movel(p[x_c + -0.047836, y_c + -0.053766, z_c, rx, ry, rz], a, v)
    movel(p[x_c + -0.047956, y_c + -0.053411, z_c, rx, ry, rz], a, v)
    movel(p[x_c + -0.048074, y_c + -0.053056, z_c, rx, ry, rz], a, v)
    movel(p[x_c + -0.048190, y_c + -0.052701, z_c, rx, ry, rz], a, v)
    movel(p[x_c + -0.048305, y_c + -0.052345, z_c, rx, ry, rz], a, v)
    movel(p[x_c + -0.048418, y_c + -0.051989, z_c, rx, ry, rz], a, v)
    movel(p[x_c + -0.048530, y_c + -0.051632, z_c, rx, ry, rz], a, v)
    movel(p[x_c + -0.048640, y_c + -0.051275, z_c, rx, ry, rz], a, v)
    movel(p[x_c + -0.048748, y_c + -0.050917, z_c, rx, ry, rz], a, v)
    movel(p[x_c + -0.048855, y_c + -0.050558, z_c, rx, ry, rz], a, v)
    movel(p[x_c + -0.048960, y_c + -0.050199, z_c, rx, ry, rz], a, v)
    movel(p[x_c + -0.049064, y_c + -0.049838, z_c, rx, ry, rz], a, v)
    movel(p[x_c + -0.049167, y_c + -0.049477, z_c, rx, ry, rz], a, v)
    movel(p[x_c + -0.049268, y_c + -0.049115, z_c, rx, ry, rz], a, v)
    movel(p[x_c + -0.049367, y_c + -0.048753, z_c, rx, ry, rz], a, v)
    movel(p[x_c + -0.049466, y_c + -0.048389, z_c, rx, ry, rz], a, v)
    movel(p[x_c + -0.049562, y_c + -0.048024, z_c, rx, ry, rz], a, v)
    movel(p[x_c + -0.049658, y_c + -0.047658, z_c, rx, ry, rz], a, v)
    movel(p[x_c + -0.049752, y_c + -0.047291, z_c, rx, ry, rz], a, v)
    movel(p[x_c + -0.049752, y_c + -0.047291, z_c, rx, ry, rz], a, v)
    movel(p[x_c + -0.050259, y_c + -0.045294, z_c, rx, ry, rz], a, v)
    movel(p[x_c + -0.050259, y_c + -0.045294, z_c, rx, ry, rz], a, v)
    movel(p[x_c + -0.050750, y_c + -0.046415, z_c, rx, ry, rz], a, v)
    movel(p[x_c + -0.050750, y_c + -0.046415, z_c, rx, ry, rz], a, v)
    movel(p[x_c + -0.050803, y_c + -0.046537, z_c, rx, ry, rz], a, v)
    movel(p[x_c + -0.050858, y_c + -0.046667, z_c, rx, ry, rz], a, v)
    movel(p[x_c + -0.050915, y_c + -0.046804, z_c, rx, ry, rz], a, v)
    movel(p[x_c + -0.050973, y_c + -0.046949, z_c, rx, ry, rz], a, v)
    movel(p[x_c + -0.051033, y_c + -0.047101, z_c, rx, ry, rz], a, v)
    movel(p[x_c + -0.051095, y_c + -0.047259, z_c, rx, ry, rz], a, v)
    movel(p[x_c + -0.051158, y_c + -0.047424, z_c, rx, ry, rz], a, v)
    movel(p[x_c + -0.051223, y_c + -0.047595, z_c, rx, ry, rz], a, v)
    movel(p[x_c + -0.051289, y_c + -0.047771, z_c, rx, ry, rz], a, v)
    movel(p[x_c + -0.051356, y_c + -0.047953, z_c, rx, ry, rz], a, v)
    movel(p[x_c + -0.051424, y_c + -0.048140, z_c, rx, ry, rz], a, v)
    movel(p[x_c + -0.051494, y_c + -0.048332, z_c, rx, ry, rz], a, v)
    movel(p[x_c + -0.051564, y_c + -0.048529, z_c, rx, ry, rz], a, v)
    movel(p[x_c + -0.051635, y_c + -0.048730, z_c, rx, ry, rz], a, v)
    movel(p[x_c + -0.051707, y_c + -0.048936, z_c, rx, ry, rz], a, v)
    movel(p[x_c + -0.051780, y_c + -0.049144, z_c, rx, ry, rz], a, v)
    movel(p[x_c + -0.051853, y_c + -0.049357, z_c, rx, ry, rz], a, v)
    movel(p[x_c + -0.051927, y_c + -0.049573, z_c, rx, ry, rz], a, v)
    movel(p[x_c + -0.052001, y_c + -0.049791, z_c, rx, ry, rz], a, v)
    movel(p[x_c + -0.052075, y_c + -0.050013, z_c, rx, ry, rz], a, v)
    movel(p[x_c + -0.052150, y_c + -0.050236, z_c, rx, ry, rz], a, v)
    movel(p[x_c + -0.052224, y_c + -0.050462, z_c, rx, ry, rz], a, v)
    movel(p[x_c + -0.052299, y_c + -0.050689, z_c, rx, ry, rz], a, v)
    movel(p[x_c + -0.052374, y_c + -0.050918, z_c, rx, ry, rz], a, v)
    movel(p[x_c + -0.052448, y_c + -0.051148, z_c, rx, ry, rz], a, v)
    movel(p[x_c + -0.052523, y_c + -0.051379, z_c, rx, ry, rz], a, v)
    movel(p[x_c + -0.052596, y_c + -0.051611, z_c, rx, ry, rz], a, v)
    movel(p[x_c + -0.052670, y_c + -0.051843, z_c, rx, ry, rz], a, v)
    movel(p[x_c + -0.052743, y_c + -0.052075, z_c, rx, ry, rz], a, v)
    movel(p[x_c + -0.052815, y_c + -0.052307, z_c, rx, ry, rz], a, v)
    movel(p[x_c + -0.052887, y_c + -0.052538, z_c, rx, ry, rz], a, v)
    movel(p[x_c + -0.052957, y_c + -0.052769, z_c, rx, ry, rz], a, v)
    movel(p[x_c + -0.053027, y_c + -0.052998, z_c, rx, ry, rz], a, v)
    movel(p[x_c + -0.053096, y_c + -0.053227, z_c, rx, ry, rz], a, v)
    movel(p[x_c + -0.053164, y_c + -0.053453, z_c, rx, ry, rz], a, v)
    movel(p[x_c + -0.053231, y_c + -0.053678, z_c, rx, ry, rz], a, v)
    movel(p[x_c + -0.053296, y_c + -0.053900, z_c, rx, ry, rz], a, v)
    movel(p[x_c + -0.053360, y_c + -0.054120, z_c, rx, ry, rz], a, v)
    movel(p[x_c + -0.053422, y_c + -0.054337, z_c, rx, ry, rz], a, v)
    movel(p[x_c + -0.053483, y_c + -0.054550, z_c, rx, ry, rz], a, v)
    movel(p[x_c + -0.053543, y_c + -0.054761, z_c, rx, ry, rz], a, v)
    movel(p[x_c + -0.053600, y_c + -0.054968, z_c, rx, ry, rz], a, v)
    movel(p[x_c + -0.053656, y_c + -0.055171, z_c, rx, ry, rz], a, v)
    movel(p[x_c + -0.053710, y_c + -0.055369, z_c, rx, ry, rz], a, v)
    movel(p[x_c + -0.053761, y_c + -0.055564, z_c, rx, ry, rz], a, v)
    movel(p[x_c + -0.053811, y_c + -0.055753, z_c, rx, ry, rz], a, v)
    movel(p[x_c + -0.053859, y_c + -0.055937, z_c, rx, ry, rz], a, v)
    movel(p[x_c + -0.053904, y_c + -0.056116, z_c, rx, ry, rz], a, v)
    movel(p[x_c + -0.053947, y_c + -0.056289, z_c, rx, ry, rz], a, v)
    movel(p[x_c + -0.053947, y_c + -0.056289, z_c, rx, ry, rz], a, v)
    movel(p[x_c + -0.053991, y_c + -0.056473, z_c, rx, ry, rz], a, v)
    movel(p[x_c + -0.054035, y_c + -0.056658, z_c, rx, ry, rz], a, v)
    movel(p[x_c + -0.054078, y_c + -0.056846, z_c, rx, ry, rz], a, v)
    movel(p[x_c + -0.054121, y_c + -0.057036, z_c, rx, ry, rz], a, v)
    movel(p[x_c + -0.054163, y_c + -0.057228, z_c, rx, ry, rz], a, v)
    movel(p[x_c + -0.054205, y_c + -0.057422, z_c, rx, ry, rz], a, v)
    movel(p[x_c + -0.054246, y_c + -0.057618, z_c, rx, ry, rz], a, v)
    movel(p[x_c + -0.054286, y_c + -0.057816, z_c, rx, ry, rz], a, v)
    movel(p[x_c + -0.054327, y_c + -0.058016, z_c, rx, ry, rz], a, v)
    movel(p[x_c + -0.054366, y_c + -0.058218, z_c, rx, ry, rz], a, v)
    movel(p[x_c + -0.054405, y_c + -0.058422, z_c, rx, ry, rz], a, v)
    movel(p[x_c + -0.054444, y_c + -0.058628, z_c, rx, ry, rz], a, v)
    movel(p[x_c + -0.054482, y_c + -0.058835, z_c, rx, ry, rz], a, v)
    movel(p[x_c + -0.054519, y_c + -0.059044, z_c, rx, ry, rz], a, v)
    movel(p[x_c + -0.054556, y_c + -0.059254, z_c, rx, ry, rz], a, v)
    movel(p[x_c + -0.054592, y_c + -0.059467, z_c, rx, ry, rz], a, v)
    movel(p[x_c + -0.054628, y_c + -0.059680, z_c, rx, ry, rz], a, v)
    movel(p[x_c + -0.054663, y_c + -0.059896, z_c, rx, ry, rz], a, v)
    movel(p[x_c + -0.054697, y_c + -0.060112, z_c, rx, ry, rz], a, v)
    movel(p[x_c + -0.054731, y_c + -0.060330, z_c, rx, ry, rz], a, v)
    movel(p[x_c + -0.054764, y_c + -0.060550, z_c, rx, ry, rz], a, v)
    movel(p[x_c + -0.054797, y_c + -0.060770, z_c, rx, ry, rz], a, v)
    movel(p[x_c + -0.054829, y_c + -0.060992, z_c, rx, ry, rz], a, v)
    movel(p[x_c + -0.054860, y_c + -0.061215, z_c, rx, ry, rz], a, v)
    movel(p[x_c + -0.054891, y_c + -0.061439, z_c, rx, ry, rz], a, v)
    movel(p[x_c + -0.054921, y_c + -0.061665, z_c, rx, ry, rz], a, v)
    movel(p[x_c + -0.054950, y_c + -0.061891, z_c, rx, ry, rz], a, v)
    movel(p[x_c + -0.054979, y_c + -0.062118, z_c, rx, ry, rz], a, v)
    movel(p[x_c + -0.055007, y_c + -0.062347, z_c, rx, ry, rz], a, v)
    movel(p[x_c + -0.055034, y_c + -0.062576, z_c, rx, ry, rz], a, v)
    movel(p[x_c + -0.055061, y_c + -0.062806, z_c, rx, ry, rz], a, v)
    movel(p[x_c + -0.055087, y_c + -0.063037, z_c, rx, ry, rz], a, v)
    movel(p[x_c + -0.055112, y_c + -0.063268, z_c, rx, ry, rz], a, v)
    movel(p[x_c + -0.055137, y_c + -0.063501, z_c, rx, ry, rz], a, v)
    movel(p[x_c + -0.055161, y_c + -0.063734, z_c, rx, ry, rz], a, v)
    movel(p[x_c + -0.055184, y_c + -0.063967, z_c, rx, ry, rz], a, v)
    movel(p[x_c + -0.055206, y_c + -0.064201, z_c, rx, ry, rz], a, v)
    movel(p[x_c + -0.055228, y_c + -0.064436, z_c, rx, ry, rz], a, v)
    movel(p[x_c + -0.055249, y_c + -0.064671, z_c, rx, ry, rz], a, v)
    movel(p[x_c + -0.055269, y_c + -0.064906, z_c, rx, ry, rz], a, v)
    movel(p[x_c + -0.055289, y_c + -0.065142, z_c, rx, ry, rz], a, v)
    movel(p[x_c + -0.055307, y_c + -0.065378, z_c, rx, ry, rz], a, v)
    movel(p[x_c + -0.055325, y_c + -0.065614, z_c, rx, ry, rz], a, v)
    movel(p[x_c + -0.055342, y_c + -0.065851, z_c, rx, ry, rz], a, v)
    movel(p[x_c + -0.055359, y_c + -0.066087, z_c, rx, ry, rz], a, v)
    movel(p[x_c + -0.055374, y_c + -0.066324, z_c, rx, ry, rz], a, v)
    movel(p[x_c + -0.055389, y_c + -0.066561, z_c, rx, ry, rz], a, v)
    movel(p[x_c + -0.055403, y_c + -0.066798, z_c, rx, ry, rz], a, v)
    movel(p[x_c + -0.055417, y_c + -0.067035, z_c, rx, ry, rz], a, v)
    movel(p[x_c + -0.055417, y_c + -0.067035, z_c, rx, ry, rz], a, v)
    movel(p[x_c + -0.055428, y_c + -0.067241, z_c, rx, ry, rz], a, v)
    movel(p[x_c + -0.055440, y_c + -0.067442, z_c, rx, ry, rz], a, v)
    movel(p[x_c + -0.055453, y_c + -0.067637, z_c, rx, ry, rz], a, v)
    movel(p[x_c + -0.055466, y_c + -0.067828, z_c, rx, ry, rz], a, v)
    movel(p[x_c + -0.055479, y_c + -0.068013, z_c, rx, ry, rz], a, v)
    movel(p[x_c + -0.055493, y_c + -0.068194, z_c, rx, ry, rz], a, v)
    movel(p[x_c + -0.055508, y_c + -0.068369, z_c, rx, ry, rz], a, v)
    movel(p[x_c + -0.055523, y_c + -0.068540, z_c, rx, ry, rz], a, v)
    movel(p[x_c + -0.055539, y_c + -0.068707, z_c, rx, ry, rz], a, v)
    movel(p[x_c + -0.055556, y_c + -0.068868, z_c, rx, ry, rz], a, v)
    movel(p[x_c + -0.055574, y_c + -0.069025, z_c, rx, ry, rz], a, v)
    movel(p[x_c + -0.055592, y_c + -0.069178, z_c, rx, ry, rz], a, v)
    movel(p[x_c + -0.055611, y_c + -0.069327, z_c, rx, ry, rz], a, v)
    movel(p[x_c + -0.055630, y_c + -0.069471, z_c, rx, ry, rz], a, v)
    movel(p[x_c + -0.055651, y_c + -0.069612, z_c, rx, ry, rz], a, v)
    movel(p[x_c + -0.055673, y_c + -0.069748, z_c, rx, ry, rz], a, v)
    movel(p[x_c + -0.055695, y_c + -0.069880, z_c, rx, ry, rz], a, v)
    movel(p[x_c + -0.055718, y_c + -0.070009, z_c, rx, ry, rz], a, v)
    movel(p[x_c + -0.055742, y_c + -0.070134, z_c, rx, ry, rz], a, v)
    movel(p[x_c + -0.055768, y_c + -0.070256, z_c, rx, ry, rz], a, v)
    movel(p[x_c + -0.055794, y_c + -0.070374, z_c, rx, ry, rz], a, v)
    movel(p[x_c + -0.055821, y_c + -0.070488, z_c, rx, ry, rz], a, v)
    movel(p[x_c + -0.055849, y_c + -0.070600, z_c, rx, ry, rz], a, v)
    movel(p[x_c + -0.055879, y_c + -0.070708, z_c, rx, ry, rz], a, v)
    movel(p[x_c + -0.055909, y_c + -0.070813, z_c, rx, ry, rz], a, v)
    movel(p[x_c + -0.055941, y_c + -0.070915, z_c, rx, ry, rz], a, v)
    movel(p[x_c + -0.055974, y_c + -0.071014, z_c, rx, ry, rz], a, v)
    movel(p[x_c + -0.056008, y_c + -0.071111, z_c, rx, ry, rz], a, v)
    movel(p[x_c + -0.056043, y_c + -0.071205, z_c, rx, ry, rz], a, v)
    movel(p[x_c + -0.056080, y_c + -0.071296, z_c, rx, ry, rz], a, v)
    movel(p[x_c + -0.056118, y_c + -0.071385, z_c, rx, ry, rz], a, v)
    movel(p[x_c + -0.056157, y_c + -0.071471, z_c, rx, ry, rz], a, v)
    movel(p[x_c + -0.056197, y_c + -0.071555, z_c, rx, ry, rz], a, v)
    movel(p[x_c + -0.056239, y_c + -0.071637, z_c, rx, ry, rz], a, v)
    movel(p[x_c + -0.056283, y_c + -0.071717, z_c, rx, ry, rz], a, v)
    movel(p[x_c + -0.056327, y_c + -0.071794, z_c, rx, ry, rz], a, v)
    movel(p[x_c + -0.056374, y_c + -0.071870, z_c, rx, ry, rz], a, v)
    movel(p[x_c + -0.056421, y_c + -0.071944, z_c, rx, ry, rz], a, v)
    movel(p[x_c + -0.056471, y_c + -0.072017, z_c, rx, ry, rz], a, v)
    movel(p[x_c + -0.056521, y_c + -0.072087, z_c, rx, ry, rz], a, v)
    movel(p[x_c + -0.056574, y_c + -0.072157, z_c, rx, ry, rz], a, v)
    movel(p[x_c + -0.056628, y_c + -0.072224, z_c, rx, ry, rz], a, v)
    movel(p[x_c + -0.056683, y_c + -0.072291, z_c, rx, ry, rz], a, v)
    movel(p[x_c + -0.056741, y_c + -0.072356, z_c, rx, ry, rz], a, v)
    movel(p[x_c + -0.056800, y_c + -0.072421, z_c, rx, ry, rz], a, v)
    movel(p[x_c + -0.056860, y_c + -0.072484, z_c, rx, ry, rz], a, v)
    movel(p[x_c + -0.056923, y_c + -0.072546, z_c, rx, ry, rz], a, v)
    movel(p[x_c + -0.056987, y_c + -0.072608, z_c, rx, ry, rz], a, v)
    movel(p[x_c + -0.057053, y_c + -0.072668, z_c, rx, ry, rz], a, v)
    movel(p[x_c + -0.057053, y_c + -0.072668, z_c, rx, ry, rz], a, v)
    movel(p[x_c + -0.057204, y_c + -0.072799, z_c, rx, ry, rz], a, v)
    movel(p[x_c + -0.057356, y_c + -0.072920, z_c, rx, ry, rz], a, v)
    movel(p[x_c + -0.057511, y_c + -0.073032, z_c, rx, ry, rz], a, v)
    movel(p[x_c + -0.057667, y_c + -0.073134, z_c, rx, ry, rz], a, v)
    movel(p[x_c + -0.057825, y_c + -0.073227, z_c, rx, ry, rz], a, v)
    movel(p[x_c + -0.057984, y_c + -0.073310, z_c, rx, ry, rz], a, v)
    movel(p[x_c + -0.058145, y_c + -0.073384, z_c, rx, ry, rz], a, v)
    movel(p[x_c + -0.058308, y_c + -0.073448, z_c, rx, ry, rz], a, v)
    movel(p[x_c + -0.058473, y_c + -0.073503, z_c, rx, ry, rz], a, v)
    movel(p[x_c + -0.058639, y_c + -0.073548, z_c, rx, ry, rz], a, v)
    movel(p[x_c + -0.058806, y_c + -0.073584, z_c, rx, ry, rz], a, v)
    movel(p[x_c + -0.058975, y_c + -0.073610, z_c, rx, ry, rz], a, v)
    movel(p[x_c + -0.059146, y_c + -0.073627, z_c, rx, ry, rz], a, v)
    movel(p[x_c + -0.059318, y_c + -0.073635, z_c, rx, ry, rz], a, v)
    movel(p[x_c + -0.059492, y_c + -0.073633, z_c, rx, ry, rz], a, v)
    movel(p[x_c + -0.059667, y_c + -0.073622, z_c, rx, ry, rz], a, v)
    movel(p[x_c + -0.059843, y_c + -0.073602, z_c, rx, ry, rz], a, v)
    movel(p[x_c + -0.060021, y_c + -0.073572, z_c, rx, ry, rz], a, v)
    movel(p[x_c + -0.060200, y_c + -0.073532, z_c, rx, ry, rz], a, v)
    movel(p[x_c + -0.060381, y_c + -0.073484, z_c, rx, ry, rz], a, v)
    movel(p[x_c + -0.060563, y_c + -0.073426, z_c, rx, ry, rz], a, v)
    movel(p[x_c + -0.060746, y_c + -0.073359, z_c, rx, ry, rz], a, v)
    movel(p[x_c + -0.060931, y_c + -0.073282, z_c, rx, ry, rz], a, v)
    movel(p[x_c + -0.061116, y_c + -0.073196, z_c, rx, ry, rz], a, v)
    movel(p[x_c + -0.061304, y_c + -0.073101, z_c, rx, ry, rz], a, v)
    movel(p[x_c + -0.061492, y_c + -0.072997, z_c, rx, ry, rz], a, v)
    movel(p[x_c + -0.061681, y_c + -0.072883, z_c, rx, ry, rz], a, v)
    movel(p[x_c + -0.061872, y_c + -0.072760, z_c, rx, ry, rz], a, v)
    movel(p[x_c + -0.062064, y_c + -0.072628, z_c, rx, ry, rz], a, v)
    movel(p[x_c + -0.062257, y_c + -0.072487, z_c, rx, ry, rz], a, v)
    movel(p[x_c + -0.062451, y_c + -0.072336, z_c, rx, ry, rz], a, v)
    movel(p[x_c + -0.062646, y_c + -0.072176, z_c, rx, ry, rz], a, v)
    movel(p[x_c + -0.062843, y_c + -0.072007, z_c, rx, ry, rz], a, v)
    movel(p[x_c + -0.063040, y_c + -0.071829, z_c, rx, ry, rz], a, v)
    movel(p[x_c + -0.063239, y_c + -0.071642, z_c, rx, ry, rz], a, v)
    movel(p[x_c + -0.063438, y_c + -0.071445, z_c, rx, ry, rz], a, v)
    movel(p[x_c + -0.063638, y_c + -0.071240, z_c, rx, ry, rz], a, v)
    movel(p[x_c + -0.063840, y_c + -0.071025, z_c, rx, ry, rz], a, v)
    movel(p[x_c + -0.064042, y_c + -0.070801, z_c, rx, ry, rz], a, v)
    movel(p[x_c + -0.064245, y_c + -0.070568, z_c, rx, ry, rz], a, v)
    movel(p[x_c + -0.064449, y_c + -0.070326, z_c, rx, ry, rz], a, v)
    movel(p[x_c + -0.064654, y_c + -0.070075, z_c, rx, ry, rz], a, v)
    movel(p[x_c + -0.064860, y_c + -0.069815, z_c, rx, ry, rz], a, v)
    movel(p[x_c + -0.065067, y_c + -0.069545, z_c, rx, ry, rz], a, v)
    movel(p[x_c + -0.065274, y_c + -0.069267, z_c, rx, ry, rz], a, v)
    movel(p[x_c + -0.065483, y_c + -0.068979, z_c, rx, ry, rz], a, v)
    movel(p[x_c + -0.065692, y_c + -0.068683, z_c, rx, ry, rz], a, v)
    movel(p[x_c + -0.065901, y_c + -0.068377, z_c, rx, ry, rz], a, v)
    movel(p[x_c + -0.066112, y_c + -0.068063, z_c, rx, ry, rz], a, v)
    movel(p[x_c + -0.066112, y_c + -0.068063, z_c, rx, ry, rz], a, v)
    movel(p[x_c + -0.066282, y_c + -0.067803, z_c, rx, ry, rz], a, v)
    movel(p[x_c + -0.066450, y_c + -0.067541, z_c, rx, ry, rz], a, v)
    movel(p[x_c + -0.066615, y_c + -0.067277, z_c, rx, ry, rz], a, v)
    movel(p[x_c + -0.066778, y_c + -0.067011, z_c, rx, ry, rz], a, v)
    movel(p[x_c + -0.066939, y_c + -0.066743, z_c, rx, ry, rz], a, v)
    movel(p[x_c + -0.067097, y_c + -0.066473, z_c, rx, ry, rz], a, v)
    movel(p[x_c + -0.067253, y_c + -0.066201, z_c, rx, ry, rz], a, v)
    movel(p[x_c + -0.067406, y_c + -0.065927, z_c, rx, ry, rz], a, v)
    movel(p[x_c + -0.067558, y_c + -0.065651, z_c, rx, ry, rz], a, v)
    movel(p[x_c + -0.067706, y_c + -0.065373, z_c, rx, ry, rz], a, v)
    movel(p[x_c + -0.067853, y_c + -0.065093, z_c, rx, ry, rz], a, v)
    movel(p[x_c + -0.067997, y_c + -0.064810, z_c, rx, ry, rz], a, v)
    movel(p[x_c + -0.068139, y_c + -0.064525, z_c, rx, ry, rz], a, v)
    movel(p[x_c + -0.068279, y_c + -0.064238, z_c, rx, ry, rz], a, v)
    movel(p[x_c + -0.068416, y_c + -0.063948, z_c, rx, ry, rz], a, v)
    movel(p[x_c + -0.068551, y_c + -0.063656, z_c, rx, ry, rz], a, v)
    movel(p[x_c + -0.068684, y_c + -0.063362, z_c, rx, ry, rz], a, v)
    movel(p[x_c + -0.068815, y_c + -0.063065, z_c, rx, ry, rz], a, v)
    movel(p[x_c + -0.068944, y_c + -0.062766, z_c, rx, ry, rz], a, v)
    movel(p[x_c + -0.069070, y_c + -0.062464, z_c, rx, ry, rz], a, v)
    movel(p[x_c + -0.069194, y_c + -0.062159, z_c, rx, ry, rz], a, v)
    movel(p[x_c + -0.069316, y_c + -0.061852, z_c, rx, ry, rz], a, v)
    movel(p[x_c + -0.069436, y_c + -0.061542, z_c, rx, ry, rz], a, v)
    movel(p[x_c + -0.069554, y_c + -0.061230, z_c, rx, ry, rz], a, v)
    movel(p[x_c + -0.069670, y_c + -0.060914, z_c, rx, ry, rz], a, v)
    movel(p[x_c + -0.069784, y_c + -0.060596, z_c, rx, ry, rz], a, v)
    movel(p[x_c + -0.069895, y_c + -0.060275, z_c, rx, ry, rz], a, v)
    movel(p[x_c + -0.070005, y_c + -0.059951, z_c, rx, ry, rz], a, v)
    movel(p[x_c + -0.070112, y_c + -0.059624, z_c, rx, ry, rz], a, v)
    movel(p[x_c + -0.070218, y_c + -0.059295, z_c, rx, ry, rz], a, v)
    movel(p[x_c + -0.070321, y_c + -0.058962, z_c, rx, ry, rz], a, v)
    movel(p[x_c + -0.070423, y_c + -0.058626, z_c, rx, ry, rz], a, v)
    movel(p[x_c + -0.070522, y_c + -0.058287, z_c, rx, ry, rz], a, v)
    movel(p[x_c + -0.070620, y_c + -0.057945, z_c, rx, ry, rz], a, v)
    movel(p[x_c + -0.070715, y_c + -0.057600, z_c, rx, ry, rz], a, v)
    movel(p[x_c + -0.070809, y_c + -0.057252, z_c, rx, ry, rz], a, v)
    movel(p[x_c + -0.070900, y_c + -0.056900, z_c, rx, ry, rz], a, v)
    movel(p[x_c + -0.070990, y_c + -0.056545, z_c, rx, ry, rz], a, v)
    movel(p[x_c + -0.071078, y_c + -0.056187, z_c, rx, ry, rz], a, v)
    movel(p[x_c + -0.071164, y_c + -0.055825, z_c, rx, ry, rz], a, v)
    movel(p[x_c + -0.071248, y_c + -0.055460, z_c, rx, ry, rz], a, v)
    movel(p[x_c + -0.071331, y_c + -0.055092, z_c, rx, ry, rz], a, v)
    movel(p[x_c + -0.071411, y_c + -0.054720, z_c, rx, ry, rz], a, v)
    movel(p[x_c + -0.071490, y_c + -0.054345, z_c, rx, ry, rz], a, v)
    movel(p[x_c + -0.071567, y_c + -0.053966, z_c, rx, ry, rz], a, v)
    movel(p[x_c + -0.071642, y_c + -0.053583, z_c, rx, ry, rz], a, v)
    movel(p[x_c + -0.071715, y_c + -0.053197, z_c, rx, ry, rz], a, v)
    movel(p[x_c + -0.071787, y_c + -0.052807, z_c, rx, ry, rz], a, v)
    movel(p[x_c + -0.071856, y_c + -0.052413, z_c, rx, ry, rz], a, v)
    movel(p[x_c + -0.071856, y_c + -0.052413, z_c, rx, ry, rz], a, v)
    movel(p[x_c + -0.071891, y_c + -0.052206, z_c, rx, ry, rz], a, v)
    movel(p[x_c + -0.071924, y_c + -0.051986, z_c, rx, ry, rz], a, v)
    movel(p[x_c + -0.071957, y_c + -0.051753, z_c, rx, ry, rz], a, v)
    movel(p[x_c + -0.071989, y_c + -0.051508, z_c, rx, ry, rz], a, v)
    movel(p[x_c + -0.072020, y_c + -0.051251, z_c, rx, ry, rz], a, v)
    movel(p[x_c + -0.072050, y_c + -0.050983, z_c, rx, ry, rz], a, v)
    movel(p[x_c + -0.072079, y_c + -0.050704, z_c, rx, ry, rz], a, v)
    movel(p[x_c + -0.072107, y_c + -0.050415, z_c, rx, ry, rz], a, v)
    movel(p[x_c + -0.072134, y_c + -0.050116, z_c, rx, ry, rz], a, v)
    movel(p[x_c + -0.072160, y_c + -0.049808, z_c, rx, ry, rz], a, v)
    movel(p[x_c + -0.072186, y_c + -0.049491, z_c, rx, ry, rz], a, v)
    movel(p[x_c + -0.072210, y_c + -0.049167, z_c, rx, ry, rz], a, v)
    movel(p[x_c + -0.072233, y_c + -0.048834, z_c, rx, ry, rz], a, v)
    movel(p[x_c + -0.072256, y_c + -0.048495, z_c, rx, ry, rz], a, v)
    movel(p[x_c + -0.072277, y_c + -0.048149, z_c, rx, ry, rz], a, v)
    movel(p[x_c + -0.072297, y_c + -0.047798, z_c, rx, ry, rz], a, v)
    movel(p[x_c + -0.072316, y_c + -0.047441, z_c, rx, ry, rz], a, v)
    movel(p[x_c + -0.072334, y_c + -0.047079, z_c, rx, ry, rz], a, v)
    movel(p[x_c + -0.072351, y_c + -0.046712, z_c, rx, ry, rz], a, v)
    movel(p[x_c + -0.072367, y_c + -0.046342, z_c, rx, ry, rz], a, v)
    movel(p[x_c + -0.072382, y_c + -0.045968, z_c, rx, ry, rz], a, v)
    movel(p[x_c + -0.072395, y_c + -0.045592, z_c, rx, ry, rz], a, v)
    movel(p[x_c + -0.072408, y_c + -0.045213, z_c, rx, ry, rz], a, v)
    movel(p[x_c + -0.072419, y_c + -0.044833, z_c, rx, ry, rz], a, v)
    movel(p[x_c + -0.072429, y_c + -0.044451, z_c, rx, ry, rz], a, v)
    movel(p[x_c + -0.072438, y_c + -0.044069, z_c, rx, ry, rz], a, v)
    movel(p[x_c + -0.072446, y_c + -0.043687, z_c, rx, ry, rz], a, v)
    movel(p[x_c + -0.072452, y_c + -0.043305, z_c, rx, ry, rz], a, v)
    movel(p[x_c + -0.072458, y_c + -0.042924, z_c, rx, ry, rz], a, v)
    movel(p[x_c + -0.072462, y_c + -0.042544, z_c, rx, ry, rz], a, v)
    movel(p[x_c + -0.072465, y_c + -0.042166, z_c, rx, ry, rz], a, v)
    movel(p[x_c + -0.072466, y_c + -0.041791, z_c, rx, ry, rz], a, v)
    movel(p[x_c + -0.072466, y_c + -0.041419, z_c, rx, ry, rz], a, v)
    movel(p[x_c + -0.072465, y_c + -0.041051, z_c, rx, ry, rz], a, v)
    movel(p[x_c + -0.072463, y_c + -0.040686, z_c, rx, ry, rz], a, v)
    movel(p[x_c + -0.072459, y_c + -0.040326, z_c, rx, ry, rz], a, v)
    movel(p[x_c + -0.072454, y_c + -0.039971, z_c, rx, ry, rz], a, v)
    movel(p[x_c + -0.072448, y_c + -0.039622, z_c, rx, ry, rz], a, v)
    movel(p[x_c + -0.072440, y_c + -0.039279, z_c, rx, ry, rz], a, v)
    movel(p[x_c + -0.072431, y_c + -0.038943, z_c, rx, ry, rz], a, v)
    movel(p[x_c + -0.072420, y_c + -0.038614, z_c, rx, ry, rz], a, v)
    movel(p[x_c + -0.072408, y_c + -0.038293, z_c, rx, ry, rz], a, v)
    movel(p[x_c + -0.072395, y_c + -0.037981, z_c, rx, ry, rz], a, v)
    movel(p[x_c + -0.072380, y_c + -0.037677, z_c, rx, ry, rz], a, v)
    movel(p[x_c + -0.072364, y_c + -0.037382, z_c, rx, ry, rz], a, v)
    movel(p[x_c + -0.072346, y_c + -0.037098, z_c, rx, ry, rz], a, v)
    movel(p[x_c + -0.072327, y_c + -0.036823, z_c, rx, ry, rz], a, v)
    movel(p[x_c + -0.072306, y_c + -0.036560, z_c, rx, ry, rz], a, v)
    movel(p[x_c + -0.072284, y_c + -0.036308, z_c, rx, ry, rz], a, v)
    movel(p[x_c + -0.072284, y_c + -0.036308, z_c, rx, ry, rz], a, v)
    movel(p[x_c + -0.072209, y_c + -0.035551, z_c, rx, ry, rz], a, v)
    movel(p[x_c + -0.072125, y_c + -0.034788, z_c, rx, ry, rz], a, v)
    movel(p[x_c + -0.072033, y_c + -0.034019, z_c, rx, ry, rz], a, v)
    movel(p[x_c + -0.071932, y_c + -0.033244, z_c, rx, ry, rz], a, v)
    movel(p[x_c + -0.071822, y_c + -0.032464, z_c, rx, ry, rz], a, v)
    movel(p[x_c + -0.071704, y_c + -0.031679, z_c, rx, ry, rz], a, v)
    movel(p[x_c + -0.071577, y_c + -0.030890, z_c, rx, ry, rz], a, v)
    movel(p[x_c + -0.071442, y_c + -0.030096, z_c, rx, ry, rz], a, v)
    movel(p[x_c + -0.071299, y_c + -0.029297, z_c, rx, ry, rz], a, v)
    movel(p[x_c + -0.071147, y_c + -0.028495, z_c, rx, ry, rz], a, v)
    movel(p[x_c + -0.070988, y_c + -0.027689, z_c, rx, ry, rz], a, v)
    movel(p[x_c + -0.070820, y_c + -0.026880, z_c, rx, ry, rz], a, v)
    movel(p[x_c + -0.070645, y_c + -0.026067, z_c, rx, ry, rz], a, v)
    movel(p[x_c + -0.070462, y_c + -0.025252, z_c, rx, ry, rz], a, v)
    movel(p[x_c + -0.070271, y_c + -0.024433, z_c, rx, ry, rz], a, v)
    movel(p[x_c + -0.070072, y_c + -0.023613, z_c, rx, ry, rz], a, v)
    movel(p[x_c + -0.069866, y_c + -0.022790, z_c, rx, ry, rz], a, v)
    movel(p[x_c + -0.069652, y_c + -0.021966, z_c, rx, ry, rz], a, v)
    movel(p[x_c + -0.069431, y_c + -0.021140, z_c, rx, ry, rz], a, v)
    movel(p[x_c + -0.069202, y_c + -0.020313, z_c, rx, ry, rz], a, v)
    movel(p[x_c + -0.068967, y_c + -0.019485, z_c, rx, ry, rz], a, v)
    movel(p[x_c + -0.068724, y_c + -0.018655, z_c, rx, ry, rz], a, v)
    movel(p[x_c + -0.068474, y_c + -0.017826, z_c, rx, ry, rz], a, v)
    movel(p[x_c + -0.068217, y_c + -0.016996, z_c, rx, ry, rz], a, v)
    movel(p[x_c + -0.067953, y_c + -0.016166, z_c, rx, ry, rz], a, v)
    movel(p[x_c + -0.067683, y_c + -0.015337, z_c, rx, ry, rz], a, v)
    movel(p[x_c + -0.067406, y_c + -0.014507, z_c, rx, ry, rz], a, v)
    movel(p[x_c + -0.067122, y_c + -0.013679, z_c, rx, ry, rz], a, v)
    movel(p[x_c + -0.066831, y_c + -0.012852, z_c, rx, ry, rz], a, v)
    movel(p[x_c + -0.066534, y_c + -0.012026, z_c, rx, ry, rz], a, v)
    movel(p[x_c + -0.066231, y_c + -0.011202, z_c, rx, ry, rz], a, v)
    movel(p[x_c + -0.065921, y_c + -0.010380, z_c, rx, ry, rz], a, v)
    movel(p[x_c + -0.065605, y_c + -0.009559, z_c, rx, ry, rz], a, v)
    movel(p[x_c + -0.065283, y_c + -0.008741, z_c, rx, ry, rz], a, v)
    movel(p[x_c + -0.064955, y_c + -0.007926, z_c, rx, ry, rz], a, v)
    movel(p[x_c + -0.064620, y_c + -0.007114, z_c, rx, ry, rz], a, v)
    movel(p[x_c + -0.064280, y_c + -0.006305, z_c, rx, ry, rz], a, v)
    movel(p[x_c + -0.063935, y_c + -0.005499, z_c, rx, ry, rz], a, v)
    movel(p[x_c + -0.063583, y_c + -0.004697, z_c, rx, ry, rz], a, v)
    movel(p[x_c + -0.063226, y_c + -0.003899, z_c, rx, ry, rz], a, v)
    movel(p[x_c + -0.062863, y_c + -0.003105, z_c, rx, ry, rz], a, v)
    movel(p[x_c + -0.062495, y_c + -0.002316, z_c, rx, ry, rz], a, v)
    movel(p[x_c + -0.062121, y_c + -0.001532, z_c, rx, ry, rz], a, v)
    movel(p[x_c + -0.061742, y_c + -0.000752, z_c, rx, ry, rz], a, v)
    movel(p[x_c + -0.061358, y_c + 0.000022, z_c, rx, ry, rz], a, v)
    movel(p[x_c + -0.060969, y_c + 0.000791, z_c, rx, ry, rz], a, v)
    movel(p[x_c + -0.060574, y_c + 0.001553, z_c, rx, ry, rz], a, v)
    movel(p[x_c + -0.060175, y_c + 0.002310, z_c, rx, ry, rz], a, v)
    movel(p[x_c + -0.059771, y_c + 0.003061, z_c, rx, ry, rz], a, v)
    movel(p[x_c + -0.059771, y_c + 0.003061, z_c, rx, ry, rz], a, v)
    movel(p[x_c + -0.058251, y_c + 0.005851, z_c, rx, ry, rz], a, v)
    movel(p[x_c + -0.058251, y_c + 0.005851, z_c, rx, ry, rz], a, v)
    movel(p[x_c + -0.058470, y_c + 0.008306, z_c, rx, ry, rz], a, v)
    movel(p[x_c + -0.058470, y_c + 0.008306, z_c, rx, ry, rz], a, v)
    movel(p[x_c + -0.058489, y_c + 0.008540, z_c, rx, ry, rz], a, v)
    movel(p[x_c + -0.058507, y_c + 0.008797, z_c, rx, ry, rz], a, v)
    movel(p[x_c + -0.058524, y_c + 0.009075, z_c, rx, ry, rz], a, v)
    movel(p[x_c + -0.058539, y_c + 0.009375, z_c, rx, ry, rz], a, v)
    movel(p[x_c + -0.058552, y_c + 0.009694, z_c, rx, ry, rz], a, v)
    movel(p[x_c + -0.058565, y_c + 0.010032, z_c, rx, ry, rz], a, v)
    movel(p[x_c + -0.058576, y_c + 0.010388, z_c, rx, ry, rz], a, v)
    movel(p[x_c + -0.058585, y_c + 0.010761, z_c, rx, ry, rz], a, v)
    movel(p[x_c + -0.058594, y_c + 0.011150, z_c, rx, ry, rz], a, v)
    movel(p[x_c + -0.058601, y_c + 0.011554, z_c, rx, ry, rz], a, v)
    movel(p[x_c + -0.058607, y_c + 0.011971, z_c, rx, ry, rz], a, v)
    movel(p[x_c + -0.058612, y_c + 0.012403, z_c, rx, ry, rz], a, v)
    movel(p[x_c + -0.058616, y_c + 0.012846, z_c, rx, ry, rz], a, v)
    movel(p[x_c + -0.058618, y_c + 0.013300, z_c, rx, ry, rz], a, v)
    movel(p[x_c + -0.058620, y_c + 0.013765, z_c, rx, ry, rz], a, v)
    movel(p[x_c + -0.058620, y_c + 0.014239, z_c, rx, ry, rz], a, v)
    movel(p[x_c + -0.058619, y_c + 0.014721, z_c, rx, ry, rz], a, v)
    movel(p[x_c + -0.058617, y_c + 0.015210, z_c, rx, ry, rz], a, v)
    movel(p[x_c + -0.058614, y_c + 0.015706, z_c, rx, ry, rz], a, v)
    movel(p[x_c + -0.058610, y_c + 0.016207, z_c, rx, ry, rz], a, v)
    movel(p[x_c + -0.058604, y_c + 0.016712, z_c, rx, ry, rz], a, v)
    movel(p[x_c + -0.058598, y_c + 0.017221, z_c, rx, ry, rz], a, v)
    movel(p[x_c + -0.058591, y_c + 0.017733, z_c, rx, ry, rz], a, v)
    movel(p[x_c + -0.058583, y_c + 0.018245, z_c, rx, ry, rz], a, v)
    movel(p[x_c + -0.058573, y_c + 0.018759, z_c, rx, ry, rz], a, v)
    movel(p[x_c + -0.058563, y_c + 0.019272, z_c, rx, ry, rz], a, v)
    movel(p[x_c + -0.058552, y_c + 0.019783, z_c, rx, ry, rz], a, v)
    movel(p[x_c + -0.058540, y_c + 0.020293, z_c, rx, ry, rz], a, v)
    movel(p[x_c + -0.058527, y_c + 0.020799, z_c, rx, ry, rz], a, v)
    movel(p[x_c + -0.058513, y_c + 0.021300, z_c, rx, ry, rz], a, v)
    movel(p[x_c + -0.058498, y_c + 0.021797, z_c, rx, ry, rz], a, v)
    movel(p[x_c + -0.058483, y_c + 0.022287, z_c, rx, ry, rz], a, v)
    movel(p[x_c + -0.058466, y_c + 0.022770, z_c, rx, ry, rz], a, v)
    movel(p[x_c + -0.058449, y_c + 0.023245, z_c, rx, ry, rz], a, v)
    movel(p[x_c + -0.058431, y_c + 0.023710, z_c, rx, ry, rz], a, v)
    movel(p[x_c + -0.058412, y_c + 0.024166, z_c, rx, ry, rz], a, v)
    movel(p[x_c + -0.058392, y_c + 0.024611, z_c, rx, ry, rz], a, v)
    movel(p[x_c + -0.058372, y_c + 0.025043, z_c, rx, ry, rz], a, v)
    movel(p[x_c + -0.058350, y_c + 0.025463, z_c, rx, ry, rz], a, v)
    movel(p[x_c + -0.058329, y_c + 0.025868, z_c, rx, ry, rz], a, v)
    movel(p[x_c + -0.058306, y_c + 0.026259, z_c, rx, ry, rz], a, v)
    movel(p[x_c + -0.058283, y_c + 0.026634, z_c, rx, ry, rz], a, v)
    movel(p[x_c + -0.058259, y_c + 0.026992, z_c, rx, ry, rz], a, v)
    movel(p[x_c + -0.058234, y_c + 0.027332, z_c, rx, ry, rz], a, v)
    movel(p[x_c + -0.058209, y_c + 0.027653, z_c, rx, ry, rz], a, v)
    movel(p[x_c + -0.058183, y_c + 0.027955, z_c, rx, ry, rz], a, v)
    movel(p[x_c + -0.058157, y_c + 0.028236, z_c, rx, ry, rz], a, v)
    movel(p[x_c + -0.058130, y_c + 0.028495, z_c, rx, ry, rz], a, v)
    movel(p[x_c + -0.058102, y_c + 0.028732, z_c, rx, ry, rz], a, v)
    movel(p[x_c + -0.058102, y_c + 0.028732, z_c, rx, ry, rz], a, v)
    movel(p[x_c + -0.058023, y_c + 0.029352, z_c, rx, ry, rz], a, v)
    movel(p[x_c + -0.057941, y_c + 0.029969, z_c, rx, ry, rz], a, v)
    movel(p[x_c + -0.057855, y_c + 0.030585, z_c, rx, ry, rz], a, v)
    movel(p[x_c + -0.057766, y_c + 0.031199, z_c, rx, ry, rz], a, v)
    movel(p[x_c + -0.057673, y_c + 0.031810, z_c, rx, ry, rz], a, v)
    movel(p[x_c + -0.057576, y_c + 0.032420, z_c, rx, ry, rz], a, v)
    movel(p[x_c + -0.057476, y_c + 0.033029, z_c, rx, ry, rz], a, v)
    movel(p[x_c + -0.057372, y_c + 0.033635, z_c, rx, ry, rz], a, v)
    movel(p[x_c + -0.057264, y_c + 0.034241, z_c, rx, ry, rz], a, v)
    movel(p[x_c + -0.057153, y_c + 0.034845, z_c, rx, ry, rz], a, v)
    movel(p[x_c + -0.057037, y_c + 0.035447, z_c, rx, ry, rz], a, v)
    movel(p[x_c + -0.056918, y_c + 0.036048, z_c, rx, ry, rz], a, v)
    movel(p[x_c + -0.056795, y_c + 0.036648, z_c, rx, ry, rz], a, v)
    movel(p[x_c + -0.056669, y_c + 0.037247, z_c, rx, ry, rz], a, v)
    movel(p[x_c + -0.056538, y_c + 0.037845, z_c, rx, ry, rz], a, v)
    movel(p[x_c + -0.056403, y_c + 0.038442, z_c, rx, ry, rz], a, v)
    movel(p[x_c + -0.056265, y_c + 0.039039, z_c, rx, ry, rz], a, v)
    movel(p[x_c + -0.056123, y_c + 0.039634, z_c, rx, ry, rz], a, v)
    movel(p[x_c + -0.055976, y_c + 0.040229, z_c, rx, ry, rz], a, v)
    movel(p[x_c + -0.055826, y_c + 0.040824, z_c, rx, ry, rz], a, v)
    movel(p[x_c + -0.055671, y_c + 0.041417, z_c, rx, ry, rz], a, v)
    movel(p[x_c + -0.055513, y_c + 0.042011, z_c, rx, ry, rz], a, v)
    movel(p[x_c + -0.055350, y_c + 0.042604, z_c, rx, ry, rz], a, v)
    movel(p[x_c + -0.055184, y_c + 0.043197, z_c, rx, ry, rz], a, v)
    movel(p[x_c + -0.055013, y_c + 0.043790, z_c, rx, ry, rz], a, v)
    movel(p[x_c + -0.054838, y_c + 0.044383, z_c, rx, ry, rz], a, v)
    movel(p[x_c + -0.054659, y_c + 0.044975, z_c, rx, ry, rz], a, v)
    movel(p[x_c + -0.054475, y_c + 0.045568, z_c, rx, ry, rz], a, v)
    movel(p[x_c + -0.054288, y_c + 0.046161, z_c, rx, ry, rz], a, v)
    movel(p[x_c + -0.054096, y_c + 0.046755, z_c, rx, ry, rz], a, v)
    movel(p[x_c + -0.053900, y_c + 0.047349, z_c, rx, ry, rz], a, v)
    movel(p[x_c + -0.053700, y_c + 0.047943, z_c, rx, ry, rz], a, v)
    movel(p[x_c + -0.053495, y_c + 0.048538, z_c, rx, ry, rz], a, v)
    movel(p[x_c + -0.053286, y_c + 0.049133, z_c, rx, ry, rz], a, v)
    movel(p[x_c + -0.053073, y_c + 0.049729, z_c, rx, ry, rz], a, v)
    movel(p[x_c + -0.052855, y_c + 0.050326, z_c, rx, ry, rz], a, v)
    movel(p[x_c + -0.052633, y_c + 0.050924, z_c, rx, ry, rz], a, v)
    movel(p[x_c + -0.052406, y_c + 0.051523, z_c, rx, ry, rz], a, v)
    movel(p[x_c + -0.052175, y_c + 0.052123, z_c, rx, ry, rz], a, v)
    movel(p[x_c + -0.051940, y_c + 0.052724, z_c, rx, ry, rz], a, v)
    movel(p[x_c + -0.051700, y_c + 0.053326, z_c, rx, ry, rz], a, v)
    movel(p[x_c + -0.051455, y_c + 0.053930, z_c, rx, ry, rz], a, v)
    movel(p[x_c + -0.051206, y_c + 0.054535, z_c, rx, ry, rz], a, v)
    movel(p[x_c + -0.050952, y_c + 0.055141, z_c, rx, ry, rz], a, v)
    movel(p[x_c + -0.050694, y_c + 0.055749, z_c, rx, ry, rz], a, v)
    movel(p[x_c + -0.050430, y_c + 0.056359, z_c, rx, ry, rz], a, v)
    movel(p[x_c + -0.050163, y_c + 0.056971, z_c, rx, ry, rz], a, v)
    movel(p[x_c + -0.049890, y_c + 0.057584, z_c, rx, ry, rz], a, v)
    movel(p[x_c + -0.049613, y_c + 0.058199, z_c, rx, ry, rz], a, v)
    movel(p[x_c + -0.049613, y_c + 0.058199, z_c, rx, ry, rz], a, v)
    movel(p[x_c + -0.049463, y_c + 0.058529, z_c, rx, ry, rz], a, v)
    movel(p[x_c + -0.049315, y_c + 0.058852, z_c, rx, ry, rz], a, v)
    movel(p[x_c + -0.049167, y_c + 0.059169, z_c, rx, ry, rz], a, v)
    movel(p[x_c + -0.049021, y_c + 0.059480, z_c, rx, ry, rz], a, v)
    movel(p[x_c + -0.048876, y_c + 0.059786, z_c, rx, ry, rz], a, v)
    movel(p[x_c + -0.048732, y_c + 0.060087, z_c, rx, ry, rz], a, v)
    movel(p[x_c + -0.048588, y_c + 0.060383, z_c, rx, ry, rz], a, v)
    movel(p[x_c + -0.048445, y_c + 0.060675, z_c, rx, ry, rz], a, v)
    movel(p[x_c + -0.048302, y_c + 0.060963, z_c, rx, ry, rz], a, v)
    movel(p[x_c + -0.048158, y_c + 0.061247, z_c, rx, ry, rz], a, v)
    movel(p[x_c + -0.048014, y_c + 0.061527, z_c, rx, ry, rz], a, v)
    movel(p[x_c + -0.047869, y_c + 0.061805, z_c, rx, ry, rz], a, v)
    movel(p[x_c + -0.047724, y_c + 0.062080, z_c, rx, ry, rz], a, v)
    movel(p[x_c + -0.047578, y_c + 0.062353, z_c, rx, ry, rz], a, v)
    movel(p[x_c + -0.047430, y_c + 0.062624, z_c, rx, ry, rz], a, v)
    movel(p[x_c + -0.047281, y_c + 0.062893, z_c, rx, ry, rz], a, v)
    movel(p[x_c + -0.047130, y_c + 0.063161, z_c, rx, ry, rz], a, v)
    movel(p[x_c + -0.046977, y_c + 0.063428, z_c, rx, ry, rz], a, v)
    movel(p[x_c + -0.046822, y_c + 0.063695, z_c, rx, ry, rz], a, v)
    movel(p[x_c + -0.046665, y_c + 0.063961, z_c, rx, ry, rz], a, v)
    movel(p[x_c + -0.046505, y_c + 0.064227, z_c, rx, ry, rz], a, v)
    movel(p[x_c + -0.046342, y_c + 0.064494, z_c, rx, ry, rz], a, v)
    movel(p[x_c + -0.046176, y_c + 0.064762, z_c, rx, ry, rz], a, v)
    movel(p[x_c + -0.046007, y_c + 0.065031, z_c, rx, ry, rz], a, v)
    movel(p[x_c + -0.045835, y_c + 0.065302, z_c, rx, ry, rz], a, v)
    movel(p[x_c + -0.045658, y_c + 0.065574, z_c, rx, ry, rz], a, v)
    movel(p[x_c + -0.045478, y_c + 0.065849, z_c, rx, ry, rz], a, v)
    movel(p[x_c + -0.045294, y_c + 0.066126, z_c, rx, ry, rz], a, v)
    movel(p[x_c + -0.045105, y_c + 0.066406, z_c, rx, ry, rz], a, v)
    movel(p[x_c + -0.044912, y_c + 0.066689, z_c, rx, ry, rz], a, v)
    movel(p[x_c + -0.044714, y_c + 0.066976, z_c, rx, ry, rz], a, v)
    movel(p[x_c + -0.044511, y_c + 0.067267, z_c, rx, ry, rz], a, v)
    movel(p[x_c + -0.044302, y_c + 0.067562, z_c, rx, ry, rz], a, v)
    movel(p[x_c + -0.044089, y_c + 0.067862, z_c, rx, ry, rz], a, v)
    movel(p[x_c + -0.043869, y_c + 0.068167, z_c, rx, ry, rz], a, v)
    movel(p[x_c + -0.043644, y_c + 0.068477, z_c, rx, ry, rz], a, v)
    movel(p[x_c + -0.043412, y_c + 0.068793, z_c, rx, ry, rz], a, v)
    movel(p[x_c + -0.043174, y_c + 0.069115, z_c, rx, ry, rz], a, v)
    movel(p[x_c + -0.042929, y_c + 0.069444, z_c, rx, ry, rz], a, v)
    movel(p[x_c + -0.042678, y_c + 0.069779, z_c, rx, ry, rz], a, v)
    movel(p[x_c + -0.042420, y_c + 0.070121, z_c, rx, ry, rz], a, v)
    movel(p[x_c + -0.042154, y_c + 0.070471, z_c, rx, ry, rz], a, v)
    movel(p[x_c + -0.041881, y_c + 0.070828, z_c, rx, ry, rz], a, v)
    movel(p[x_c + -0.041600, y_c + 0.071194, z_c, rx, ry, rz], a, v)
